LIN {X 0,Y 573.093,Z 391.869,A -85,B 0,C 180,E1 -2255.983,E2 -2255.983} C_VEL
LIN {X 0,Y 573.103,Z 385.471,A -85,B 0,C 180,E1 -2257.043,E2 -2257.043} C_VEL
LIN {X 0,Y 573.177,Z 377.482,A -85,B 0,C 180,E1 -2258.106,E2 -2258.106} C_VEL
LIN {X 0,Y 573.253,Z 369.34,A -85,B 0,C 180,E1 -2258.992,E2 -2258.992} C_VEL
LIN {X 0,Y 573.348,Z 359.406,A -85,B 0,C 180,E1 -2259.881,E2 -2259.881} C_VEL
LIN {X 0,Y 573.512,Z 348.221,A -85,B 0,C 180,E1 -2260.679,E2 -2260.679} C_VEL
LIN {X 0,Y 573.585,Z 337.185,A -85,B 0,C 180,E1 -2261.305,E2 -2261.305} C_VEL
LIN {X 0,Y 573.699,Z 324.995,A -85,B 0,C 180,E1 -2261.84,E2 -2261.84} C_VEL
LIN {X 0,Y 573.829,Z 312.198,A -85,B 0,C 180,E1 -2262.241,E2 -2262.241} C_VEL
LIN {X 0,Y 573.911,Z 300.143,A -85,B 0,C 180,E1 -2262.486,E2 -2262.486} C_VEL
LIN {X 0,Y 573.985,Z 198.766,A -85,B 0,C 180,E1 -2263.768,E2 -2263.768} C_VEL
LIN {X 0,Y 573.395,Z 194.617,A -85,B 0,C 180,E1 -2263.85,E2 -2263.85} C_VEL
LIN {X 0,Y 573.569,Z 174.135,A -85,B 0,C 180,E1 -2266.725,E2 -2266.725} C_VEL
LIN {X 0,Y 573.784,Z 153.422,A -85,B 0,C 180,E1 -2269.646,E2 -2269.646} C_VEL
LIN {X 0,Y 573.931,Z 133.412,A -85,B 0,C 180,E1 -2272.498,E2 -2272.498} C_VEL
LIN {X 0,Y 573.521,Z 128.586,A -85,B 0,C 180,E1 -2273.211,E2 -2273.211} C_VEL
LIN {X 0,Y 573.218,Z 127.086,A -85,B 0,C 180,E1 -2273.44,E2 -2273.44} C_VEL
LIN {X 0,Y 573.238,Z 127.079,A -85,B 0,C 180,E1 -2276.19,E2 -2276.19} C_VEL
LIN {X 0,Y 573.203,Z 127.08,A -85,B 0,C 180,E1 -2278.565,E2 -2278.565} C_VEL
LIN {X 0,Y 573.214,Z 127.08,A -85,B 0,C 180,E1 -2280.993,E2 -2280.993} C_VEL
LIN {X 0,Y 573.238,Z 127.084,A -85,B 0,C 180,E1 -2283.52,E2 -2283.52} C_VEL
LIN {X 0,Y 573.184,Z 127.083,A -85,B 0,C 180,E1 -2286.053,E2 -2286.053} C_VEL
LIN {X 0,Y 573.229,Z 127.077,A -85,B 0,C 180,E1 -2288.702,E2 -2288.702} C_VEL
LIN {X 0,Y 573.205,Z 127.084,A -85,B 0,C 180,E1 -2291.59,E2 -2291.59} C_VEL
LIN {X 0,Y 573.216,Z 127.077,A -85,B 0,C 180,E1 -2294.334,E2 -2294.334} C_VEL
LIN {X 0,Y 573.212,Z 127.084,A -85,B 0,C 180,E1 -2297.36,E2 -2297.36} C_VEL
LIN {X 0,Y 573.224,Z 127.077,A -85,B 0,C 180,E1 -2300.391,E2 -2300.391} C_VEL
LIN {X 0,Y 573.223,Z 127.085,A -85,B 0,C 180,E1 -2303.075,E2 -2303.075} C_VEL
LIN {X 0,Y 573.238,Z 127.075,A -85,B 0,C 180,E1 -2305.669,E2 -2305.669} C_VEL
LIN {X 0,Y 573.215,Z 127.078,A -85,B 0,C 180,E1 -2308.183,E2 -2308.183} C_VEL
LIN {X 0,Y 573.222,Z 127.084,A -85,B 0,C 180,E1 -2310.632,E2 -2310.632} C_VEL
LIN {X 0,Y 573.205,Z 127.079,A -85,B 0,C 180,E1 -2313.512,E2 -2313.512} C_VEL
LIN {X 0,Y 573.184,Z 127.084,A -85,B 0,C 180,E1 -2316.132,E2 -2316.132} C_VEL
LIN {X 0,Y 573.215,Z 127.079,A -85,B 0,C 180,E1 -2319.172,E2 -2319.172} C_VEL
LIN {X 0,Y 573.181,Z 127.082,A -85,B 0,C 180,E1 -2321.41,E2 -2321.41} C_VEL
LIN {X 0,Y 573.192,Z 127.089,A -85,B 0,C 180,E1 -2324.351,E2 -2324.351} C_VEL
LIN {X 0,Y 573.183,Z 127.088,A -85,B 0,C 180,E1 -2326.528,E2 -2326.528} C_VEL
LIN {X 0,Y 573.234,Z 127.075,A -85,B 0,C 180,E1 -2329.403,E2 -2329.403} C_VEL
LIN {X 0,Y 573.207,Z 127.087,A -85,B 0,C 180,E1 -2332.249,E2 -2332.249} C_VEL
LIN {X 0,Y 573.262,Z 127.071,A -85,B 0,C 180,E1 -2335.077,E2 -2335.077} C_VEL
LIN {X 0,Y 573.301,Z 127.074,A -85,B 0,C 180,E1 -2337.892,E2 -2337.892} C_VEL
LIN {X 0,Y 573.307,Z 127.075,A -85,B 0,C 180,E1 -2340,E2 -2340} C_VEL
LIN {X 0,Y 573.26,Z 127.072,A -85,B 0,C 180,E1 -2342.811,E2 -2342.811} C_VEL
LIN {X 0,Y 573.267,Z 127.078,A -85,B 0,C 180,E1 -2345.628,E2 -2345.628} C_VEL
LIN {X 0,Y 573.232,Z 127.076,A -85,B 0,C 180,E1 -2348.46,E2 -2348.46} C_VEL
LIN {X 0,Y 573.261,Z 127.076,A -85,B 0,C 180,E1 -2351.312,E2 -2351.312} C_VEL
LIN {X 0,Y 573.246,Z 127.074,A -85,B 0,C 180,E1 -2354.415,E2 -2354.415} C_VEL
LIN {X 0,Y 573.168,Z 127.087,A -85,B 0,C 180,E1 -2357.114,E2 -2357.114} C_VEL
LIN {X 0,Y 573.255,Z 127.081,A -85,B 0,C 180,E1 -2359.331,E2 -2359.331} C_VEL
LIN {X 0,Y 573.21,Z 127.078,A -85,B 0,C 180,E1 -2362.339,E2 -2362.339} C_VEL
LIN {X 0,Y 573.187,Z 127.081,A -85,B 0,C 180,E1 -2364.347,E2 -2364.347} C_VEL
LIN {X 0,Y 572.548,Z 127.166,A -85,B 0,C 180,E1 -2364.933,E2 -2364.933} C_VEL
LIN {X 0,Y 569.719,Z 127.523,A -85,B 0,C 180,E1 -2365.885,E2 -2365.885} C_VEL
LIN {X 0,Y 567.301,Z 127.827,A -85,B 0,C 180,E1 -2366.65,E2 -2366.65} C_VEL
LIN {X 0,Y 566.245,Z 127.955,A -85,B 0,C 180,E1 -2367.242,E2 -2367.242} C_VEL
LIN {X 0,Y 566.15,Z 127.963,A -85,B 0,C 180,E1 -2367.442,E2 -2367.442} C_VEL
LIN {X 0,Y 566.159,Z 127.958,A -85,B 0,C 180,E1 -2369.771,E2 -2369.771} C_VEL
LIN {X 0,Y 566.184,Z 127.954,A -85,B 0,C 180,E1 -2372.429,E2 -2372.429} C_VEL
LIN {X 0,Y 566.168,Z 127.965,A -85,B 0,C 180,E1 -2374.99,E2 -2374.99} C_VEL
LIN {X 0,Y 566.187,Z 127.955,A -85,B 0,C 180,E1 -2377.462,E2 -2377.462} C_VEL
LIN {X 0,Y 566.199,Z 127.953,A -85,B 0,C 180,E1 -2380.2,E2 -2380.2} C_VEL
LIN {X 0,Y 566.174,Z 127.959,A -85,B 0,C 180,E1 -2383.057,E2 -2383.057} C_VEL
LIN {X 0,Y 566.187,Z 127.954,A -85,B 0,C 180,E1 -2386.05,E2 -2386.05} C_VEL
LIN {X 0,Y 566.199,Z 127.953,A -85,B 0,C 180,E1 -2389.216,E2 -2389.216} C_VEL
LIN {X 0,Y 566.175,Z 127.954,A -85,B 0,C 180,E1 -2391.637,E2 -2391.637} C_VEL
LIN {X 0,Y 566.145,Z 127.965,A -85,B 0,C 180,E1 -2394.308,E2 -2394.308} C_VEL
LIN {X 0,Y 566.206,Z 127.953,A -85,B 0,C 180,E1 -2396.898,E2 -2396.898} C_VEL
LIN {X 0,Y 566.167,Z 127.955,A -85,B 0,C 180,E1 -2399.407,E2 -2399.407} C_VEL
LIN {X 0,Y 566.186,Z 127.957,A -85,B 0,C 180,E1 -2401.857,E2 -2401.857} C_VEL
LIN {X 0,Y 566.194,Z 127.961,A -85,B 0,C 180,E1 -2404.251,E2 -2404.251} C_VEL
LIN {X 0,Y 566.17,Z 127.956,A -85,B 0,C 180,E1 -2407.369,E2 -2407.369} C_VEL
LIN {X 0,Y 566.202,Z 127.957,A -85,B 0,C 180,E1 -2409.663,E2 -2409.663} C_VEL
LIN {X 0,Y 566.225,Z 128.065,A -85,B 0,C 180,E1 -2410.877,E2 -2410.877} C_VEL
LIN {X 0,Y 566.465,Z 134.818,A -85,B 0,C 180,E1 -2412.118,E2 -2412.118} C_VEL
LIN {X 0,Y 566.294,Z 150.062,A -85,B 0,C 180,E1 -2414.894,E2 -2414.894} C_VEL
LIN {X 0,Y 566.255,Z 156.422,A -85,B 0,C 180,E1 -2416.055,E2 -2416.055} C_VEL
LIN {X 0,Y 567.161,Z 162.399,A -85,B 0,C 180,E1 -2416.155,E2 -2416.155} C_VEL
LIN {X 0,Y 566.967,Z 262.997,A -85,B 0,C 180,E1 -2417.449,E2 -2417.449} C_VEL
LIN {X 0,Y 566.83,Z 276.241,A -85,B 0,C 180,E1 -2417.764,E2 -2417.764} C_VEL
LIN {X 0,Y 566.736,Z 288.394,A -85,B 0,C 180,E1 -2418.194,E2 -2418.194} C_VEL
LIN {X 0,Y 566.611,Z 300.586,A -85,B 0,C 180,E1 -2418.777,E2 -2418.777} C_VEL
LIN {X 0,Y 566.448,Z 311.561,A -85,B 0,C 180,E1 -2419.456,E2 -2419.456} C_VEL
LIN {X 0,Y 566.326,Z 322.078,A -85,B 0,C 180,E1 -2420.266,E2 -2420.266} C_VEL
LIN {X 0,Y 566.221,Z 330.674,A -85,B 0,C 180,E1 -2421.075,E2 -2421.075} C_VEL
LIN {X 0,Y 566.112,Z 338.594,A -85,B 0,C 180,E1 -2421.972,E2 -2421.972} C_VEL
LIN {X 0,Y 566.049,Z 345.161,A -85,B 0,C 180,E1 -2422.868,E2 -2422.868} C_VEL
LIN {X 0,Y 566.003,Z 351.63,A -85,B 0,C 180,E1 -2423.942,E2 -2423.942} C_VEL
LIN {X 0,Y 565.877,Z 356.766,A -85,B 0,C 180,E1 -2425.013,E2 -2425.013} C_VEL
LIN {X 0,Y 565.926,Z 360.755,A -85,B 0,C 180,E1 -2426.084,E2 -2426.084} C_VEL
LIN {X 0,Y 565.877,Z 363.704,A -85,B 0,C 180,E1 -2427.153,E2 -2427.153} C_VEL
LIN {X 0,Y 565.841,Z 365.127,A -85,B 0,C 180,E1 -2427.865,E2 -2427.865} C_VEL
LIN {X 0,Y 565.841,Z 366.757,A -85,B 0,C 180,E1 -2429.289,E2 -2429.289} C_VEL
LIN {X 0,Y 565.839,Z 366.996,A -85,B 0,C 180,E1 -2430,E2 -2430} C_VEL
LIN {X 0,Y 565.841,Z 366.815,A -85,B 0,C 180,E1 -2430.712,E2 -2430.712} C_VEL
LIN {X 0,Y 565.841,Z 365.266,A -85,B 0,C 180,E1 -2432.136,E2 -2432.136} C_VEL
LIN {X 0,Y 565.878,Z 363.905,A -85,B 0,C 180,E1 -2432.848,E2 -2432.848} C_VEL
LIN {X 0,Y 565.927,Z 361.028,A -85,B 0,C 180,E1 -2433.917,E2 -2433.917} C_VEL
LIN {X 0,Y 565.878,Z 357.128,A -85,B 0,C 180,E1 -2434.988,E2 -2434.988} C_VEL
LIN {X 0,Y 565.991,Z 352.096,A -85,B 0,C 180,E1 -2436.059,E2 -2436.059} C_VEL
LIN {X 0,Y 566.031,Z 345.77,A -85,B 0,C 180,E1 -2437.133,E2 -2437.133} C_VEL
LIN {X 0,Y 566.128,Z 337.847,A -85,B 0,C 180,E1 -2438.208,E2 -2438.208} C_VEL
LIN {X 0,Y 566.249,Z 327.995,A -85,B 0,C 180,E1 -2439.285,E2 -2439.285} C_VEL
LIN {X 0,Y 566.424,Z 317.675,A -85,B 0,C 180,E1 -2440.184,E2 -2440.184} C_VEL
LIN {X 0,Y 566.507,Z 306.391,A -85,B 0,C 180,E1 -2440.973,E2 -2440.973} C_VEL
LIN {X 0,Y 566.691,Z 295.182,A -85,B 0,C 180,E1 -2441.592,E2 -2441.592} C_VEL
LIN {X 0,Y 566.788,Z 282.587,A -85,B 0,C 180,E1 -2442.119,E2 -2442.119} C_VEL
LIN {X 0,Y 566.93,Z 269.409,A -85,B 0,C 180,E1 -2442.507,E2 -2442.507} C_VEL
LIN {X 0,Y 567.04,Z 257.034,A -85,B 0,C 180,E1 -2442.732,E2 -2442.732} C_VEL
LIN {X 0,Y 567.066,Z 161.334,A -85,B 0,C 180,E1 -2443.951,E2 -2443.951} C_VEL
LIN {X 0,Y 566.237,Z 156.331,A -85,B 0,C 180,E1 -2444.052,E2 -2444.052} C_VEL
LIN {X 0,Y 566.391,Z 140.839,A -85,B 0,C 180,E1 -2446.877,E2 -2446.877} C_VEL
LIN {X 0,Y 566.442,Z 130.18,A -85,B 0,C 180,E1 -2448.82,E2 -2448.82} C_VEL
LIN {X 0,Y 566.223,Z 127.955,A -85,B 0,C 180,E1 -2449.251,E2 -2449.251} C_VEL
LIN {X 0,Y 566.189,Z 127.961,A -85,B 0,C 180,E1 -2451.863,E2 -2451.863} C_VEL
LIN {X 0,Y 566.185,Z 127.954,A -85,B 0,C 180,E1 -2455.022,E2 -2455.022} C_VEL
LIN {X 0,Y 566.173,Z 127.957,A -85,B 0,C 180,E1 -2457.341,E2 -2457.341} C_VEL
LIN {X 0,Y 566.173,Z 127.964,A -85,B 0,C 180,E1 -2459.77,E2 -2459.77} C_VEL
LIN {X 0,Y 566.201,Z 127.952,A -85,B 0,C 180,E1 -2462.429,E2 -2462.429} C_VEL
LIN {X 0,Y 566.178,Z 127.955,A -85,B 0,C 180,E1 -2464.989,E2 -2464.989} C_VEL
LIN {X 0,Y 566.192,Z 127.96,A -85,B 0,C 180,E1 -2467.461,E2 -2467.461} C_VEL
LIN {X 0,Y 566.206,Z 127.951,A -85,B 0,C 180,E1 -2470.199,E2 -2470.199} C_VEL
LIN {X 0,Y 566.192,Z 127.956,A -85,B 0,C 180,E1 -2473.055,E2 -2473.055} C_VEL
LIN {X 0,Y 566.157,Z 127.957,A -85,B 0,C 180,E1 -2476.053,E2 -2476.053} C_VEL
LIN {X 0,Y 566.165,Z 127.959,A -85,B 0,C 180,E1 -2478.859,E2 -2478.859} C_VEL
LIN {X 0,Y 566.202,Z 127.956,A -85,B 0,C 180,E1 -2481.443,E2 -2481.443} C_VEL
LIN {X 0,Y 566.141,Z 127.959,A -85,B 0,C 180,E1 -2484.306,E2 -2484.306} C_VEL
LIN {X 0,Y 566.192,Z 127.96,A -85,B 0,C 180,E1 -2486.896,E2 -2486.896} C_VEL
LIN {X 0,Y 566.159,Z 127.959,A -85,B 0,C 180,E1 -2489.406,E2 -2489.406} C_VEL
LIN {X 0,Y 566.147,Z 127.958,A -85,B 0,C 180,E1 -2491.854,E2 -2491.854} C_VEL
LIN {X 0,Y 566.197,Z 127.954,A -85,B 0,C 180,E1 -2494.25,E2 -2494.25} C_VEL
LIN {X 0,Y 566.158,Z 127.958,A -85,B 0,C 180,E1 -2497.367,E2 -2497.367} C_VEL
LIN {X 0,Y 566.194,Z 127.952,A -85,B 0,C 180,E1 -2499.662,E2 -2499.662} C_VEL
LIN {X 0,Y 566.161,Z 127.957,A -85,B 0,C 180,E1 -2501.92,E2 -2501.92} C_VEL
LIN {X 0,Y 566.176,Z 127.958,A -85,B 0,C 180,E1 -2504.89,E2 -2504.89} C_VEL
LIN {X 0,Y 566.173,Z 127.956,A -85,B 0,C 180,E1 -2507.818,E2 -2507.818} C_VEL
LIN {X 0,Y 566.163,Z 127.96,A -85,B 0,C 180,E1 -2509.992,E2 -2509.992} C_VEL
LIN {X 0,Y 566.178,Z 127.956,A -85,B 0,C 180,E1 -2512.869,E2 -2512.869} C_VEL
LIN {X 0,Y 566.246,Z 127.946,A -85,B 0,C 180,E1 -2515.016,E2 -2515.016} C_VEL
LIN {X 0,Y 566.274,Z 127.947,A -85,B 0,C 180,E1 -2517.866,E2 -2517.866} C_VEL
LIN {X 0,Y 566.281,Z 127.95,A -85,B 0,C 180,E1 -2520,E2 -2520} C_VEL
LIN {X 0,Y 566.232,Z 127.947,A -85,B 0,C 180,E1 -2522.846,E2 -2522.846} C_VEL
LIN {X 0,Y 566.229,Z 127.954,A -85,B 0,C 180,E1 -2525.699,E2 -2525.699} C_VEL
LIN {X 0,Y 566.178,Z 127.955,A -85,B 0,C 180,E1 -2528.566,E2 -2528.566} C_VEL
LIN {X 0,Y 566.187,Z 127.958,A -85,B 0,C 180,E1 -2531.455,E2 -2531.455} C_VEL
LIN {X 0,Y 566.178,Z 127.954,A -85,B 0,C 180,E1 -2534.486,E2 -2534.486} C_VEL
LIN {X 0,Y 566.152,Z 127.963,A -85,B 0,C 180,E1 -2537.333,E2 -2537.333} C_VEL
LIN {X 0,Y 566.169,Z 127.964,A -85,B 0,C 180,E1 -2539.582,E2 -2539.582} C_VEL
LIN {X 0,Y 566.141,Z 127.962,A -85,B 0,C 180,E1 -2541.865,E2 -2541.865} C_VEL
LIN {X 0,Y 566.147,Z 127.958,A -85,B 0,C 180,E1 -2544.183,E2 -2544.183} C_VEL
LIN {X 0,Y 566.17,Z 127.956,A -85,B 0,C 180,E1 -2546.652,E2 -2546.652} C_VEL
LIN {X 0,Y 566.143,Z 127.96,A -85,B 0,C 180,E1 -2549.772,E2 -2549.772} C_VEL
LIN {X 0,Y 566.188,Z 127.953,A -85,B 0,C 180,E1 -2552.428,E2 -2552.428} C_VEL
LIN {X 0,Y 566.16,Z 127.964,A -85,B 0,C 180,E1 -2554.987,E2 -2554.987} C_VEL
LIN {X 0,Y 566.188,Z 127.956,A -85,B 0,C 180,E1 -2557.462,E2 -2557.462} C_VEL
LIN {X 0,Y 566.203,Z 127.952,A -85,B 0,C 180,E1 -2560.2,E2 -2560.2} C_VEL
LIN {X 0,Y 566.177,Z 127.96,A -85,B 0,C 180,E1 -2563.057,E2 -2563.057} C_VEL
LIN {X 0,Y 566.155,Z 127.958,A -85,B 0,C 180,E1 -2566.054,E2 -2566.054} C_VEL
LIN {X 0,Y 566.163,Z 127.963,A -85,B 0,C 180,E1 -2568.86,E2 -2568.86} C_VEL
LIN {X 0,Y 566.198,Z 127.952,A -85,B 0,C 180,E1 -2571.444,E2 -2571.444} C_VEL
LIN {X 0,Y 566.141,Z 127.965,A -85,B 0,C 180,E1 -2574.306,E2 -2574.306} C_VEL
LIN {X 0,Y 566.195,Z 127.955,A -85,B 0,C 180,E1 -2576.896,E2 -2576.896} C_VEL
LIN {X 0,Y 566.168,Z 127.956,A -85,B 0,C 180,E1 -2579.407,E2 -2579.407} C_VEL
LIN {X 0,Y 566.171,Z 127.959,A -85,B 0,C 180,E1 -2581.855,E2 -2581.855} C_VEL
LIN {X 0,Y 566.194,Z 127.962,A -85,B 0,C 180,E1 -2584.25,E2 -2584.25} C_VEL
LIN {X 0,Y 566.179,Z 128.025,A -85,B 0,C 180,E1 -2586.426,E2 -2586.426} C_VEL
LIN {X 0,Y 567.021,Z 133.161,A -85,B 0,C 180,E1 -2587.211,E2 -2587.211} C_VEL
LIN {X 0,Y 566.812,Z 152.9,A -85,B 0,C 180,E1 -2590.064,E2 -2590.064} C_VEL
LIN {X 0,Y 566.588,Z 174.338,A -85,B 0,C 180,E1 -2593.111,E2 -2593.111} C_VEL
LIN {X 0,Y 566.39,Z 194.612,A -85,B 0,C 180,E1 -2595.974,E2 -2595.974} C_VEL
LIN {X 0,Y 567.155,Z 200.495,A -85,B 0,C 180,E1 -2596.085,E2 -2596.085} C_VEL
LIN {X 0,Y 566.961,Z 302.936,A -85,B 0,C 180,E1 -2597.403,E2 -2597.403} C_VEL
LIN {X 0,Y 566.84,Z 316.211,A -85,B 0,C 180,E1 -2597.718,E2 -2597.718} C_VEL
LIN {X 0,Y 566.743,Z 328.373,A -85,B 0,C 180,E1 -2598.148,E2 -2598.148} C_VEL
LIN {X 0,Y 566.604,Z 340.235,A -85,B 0,C 180,E1 -2598.712,E2 -2598.712} C_VEL
LIN {X 0,Y 566.439,Z 352.192,A -85,B 0,C 180,E1 -2599.455,E2 -2599.455} C_VEL
LIN {X 0,Y 566.325,Z 362.602,A -85,B 0,C 180,E1 -2600.265,E2 -2600.265} C_VEL
LIN {X 0,Y 566.207,Z 371.111,A -85,B 0,C 180,E1 -2601.074,E2 -2601.074} C_VEL
LIN {X 0,Y 566.112,Z 378.958,A -85,B 0,C 180,E1 -2601.971,E2 -2601.971} C_VEL
LIN {X 0,Y 566.004,Z 386.621,A -85,B 0,C 180,E1 -2603.046,E2 -2603.046} C_VEL
LIN {X 0,Y 566.004,Z 393.678,A -85,B 0,C 180,E1 -2604.299,E2 -2604.299} C_VEL
LIN {X 0,Y 565.933,Z 398.371,A -85,B 0,C 180,E1 -2605.37,E2 -2605.37} C_VEL
LIN {X 0,Y 565.927,Z 401.957,A -85,B 0,C 180,E1 -2606.44,E2 -2606.44} C_VEL
LIN {X 0,Y 565.878,Z 403.807,A -85,B 0,C 180,E1 -2607.152,E2 -2607.152} C_VEL
LIN {X 0,Y 565.846,Z 406.183,A -85,B 0,C 180,E1 -2608.576,E2 -2608.576} C_VEL
LIN {X 0,Y 565.839,Z 407,A -85,B 0,C 180,E1 -2610,E2 -2610} C_VEL
LIN {X 0,Y 565.846,Z 406.185,A -85,B 0,C 180,E1 -2611.423,E2 -2611.423} C_VEL
LIN {X 0,Y 565.878,Z 403.811,A -85,B 0,C 180,E1 -2612.847,E2 -2612.847} C_VEL
LIN {X 0,Y 565.926,Z 400.897,A -85,B 0,C 180,E1 -2613.916,E2 -2613.916} C_VEL
LIN {X 0,Y 565.878,Z 396.95,A -85,B 0,C 180,E1 -2614.987,E2 -2614.987} C_VEL
LIN {X 0,Y 566.004,Z 391.87,A -85,B 0,C 180,E1 -2616.058,E2 -2616.058} C_VEL
LIN {X 0,Y 566.04,Z 385.471,A -85,B 0,C 180,E1 -2617.132,E2 -2617.132} C_VEL
LIN {X 0,Y 566.133,Z 377.482,A -85,B 0,C 180,E1 -2618.207,E2 -2618.207} C_VEL
LIN {X 0,Y 566.228,Z 369.339,A -85,B 0,C 180,E1 -2619.105,E2 -2619.105} C_VEL
LIN {X 0,Y 566.347,Z 359.405,A -85,B 0,C 180,E1 -2620.004,E2 -2620.004} C_VEL
LIN {X 0,Y 566.535,Z 348.299,A -85,B 0,C 180,E1 -2620.807,E2 -2620.807} C_VEL
LIN {X 0,Y 566.611,Z 337.183,A -85,B 0,C 180,E1 -2621.446,E2 -2621.446} C_VEL
LIN {X 0,Y 566.744,Z 324.992,A -85,B 0,C 180,E1 -2621.987,E2 -2621.987} C_VEL
LIN {X 0,Y 566.913,Z 312.197,A -85,B 0,C 180,E1 -2622.393,E2 -2622.393} C_VEL
LIN {X 0,Y 567.006,Z 300.142,A -85,B 0,C 180,E1 -2622.641,E2 -2622.641} C_VEL
LIN {X 0,Y 567.051,Z 199.325,A -85,B 0,C 180,E1 -2623.932,E2 -2623.932} C_VEL
LIN {X 0,Y 566.39,Z 194.617,A -85,B 0,C 180,E1 -2624.025,E2 -2624.025} C_VEL
LIN {X 0,Y 566.588,Z 174.314,A -85,B 0,C 180,E1 -2626.892,E2 -2626.892} C_VEL
LIN {X 0,Y 566.853,Z 151.591,A -85,B 0,C 180,E1 -2630.123,E2 -2630.123} C_VEL
LIN {X 0,Y 566.992,Z 133.166,A -85,B 0,C 180,E1 -2632.789,E2 -2632.789} C_VEL
LIN {X 0,Y 566.196,Z 127.961,A -85,B 0,C 180,E1 -2633.597,E2 -2633.597} C_VEL
LIN {X 0,Y 566.187,Z 127.955,A -85,B 0,C 180,E1 -2636.542,E2 -2636.542} C_VEL
LIN {X 0,Y 566.161,Z 127.958,A -85,B 0,C 180,E1 -2638.954,E2 -2638.954} C_VEL
LIN {X 0,Y 566.18,Z 127.961,A -85,B 0,C 180,E1 -2641.422,E2 -2641.422} C_VEL
LIN {X 0,Y 566.191,Z 127.956,A -85,B 0,C 180,E1 -2643.956,E2 -2643.956} C_VEL
LIN {X 0,Y 566.176,Z 127.954,A -85,B 0,C 180,E1 -2646.571,E2 -2646.571} C_VEL
LIN {X 0,Y 566.204,Z 127.955,A -85,B 0,C 180,E1 -2649.684,E2 -2649.684} C_VEL
LIN {X 0,Y 566.165,Z 127.956,A -85,B 0,C 180,E1 -2652.09,E2 -2652.09} C_VEL
LIN {X 0,Y 566.158,Z 127.962,A -85,B 0,C 180,E1 -2654.962,E2 -2654.962} C_VEL
LIN {X 0,Y 566.163,Z 127.956,A -85,B 0,C 180,E1 -2657.908,E2 -2657.908} C_VEL
LIN {X 0,Y 566.2,Z 127.956,A -85,B 0,C 180,E1 -2660.725,E2 -2660.725} C_VEL
LIN {X 0,Y 566.172,Z 127.958,A -85,B 0,C 180,E1 -2663.428,E2 -2663.428} C_VEL
LIN {X 0,Y 566.187,Z 127.954,A -85,B 0,C 180,E1 -2666.268,E2 -2666.268} C_VEL
LIN {X 0,Y 566.172,Z 127.963,A -85,B 0,C 180,E1 -2668.925,E2 -2668.925} C_VEL
LIN {X 0,Y 566.139,Z 127.959,A -85,B 0,C 180,E1 -2671.853,E2 -2671.853} C_VEL
LIN {X 0,Y 566.181,Z 127.957,A -85,B 0,C 180,E1 -2674.249,E2 -2674.249} C_VEL
LIN {X 0,Y 566.135,Z 127.96,A -85,B 0,C 180,E1 -2677.367,E2 -2677.367} C_VEL
LIN {X 0,Y 566.158,Z 127.957,A -85,B 0,C 180,E1 -2679.661,E2 -2679.661} C_VEL
LIN {X 0,Y 566.151,Z 127.959,A -85,B 0,C 180,E1 -2681.92,E2 -2681.92} C_VEL
LIN {X 0,Y 566.168,Z 127.958,A -85,B 0,C 180,E1 -2684.89,E2 -2684.89} C_VEL
LIN {X 0,Y 566.166,Z 127.958,A -85,B 0,C 180,E1 -2687.817,E2 -2687.817} C_VEL
LIN {X 0,Y 566.151,Z 127.963,A -85,B 0,C 180,E1 -2689.992,E2 -2689.992} C_VEL
LIN {X 0,Y 566.17,Z 127.956,A -85,B 0,C 180,E1 -2692.869,E2 -2692.869} C_VEL
LIN {X 0,Y 566.238,Z 127.947,A -85,B 0,C 180,E1 -2695.016,E2 -2695.016} C_VEL
LIN {X 0,Y 566.27,Z 127.95,A -85,B 0,C 180,E1 -2697.866,E2 -2697.866} C_VEL
LIN {X 0,Y 566.275,Z 127.951,A -85,B 0,C 180,E1 -2700,E2 -2700} C_VEL
LIN {X 0,Y 566.228,Z 127.948,A -85,B 0,C 180,E1 -2702.846,E2 -2702.846} C_VEL
LIN {X 0,Y 566.236,Z 127.955,A -85,B 0,C 180,E1 -2705.699,E2 -2705.699} C_VEL
LIN {X 0,Y 566.183,Z 127.953,A -85,B 0,C 180,E1 -2708.566,E2 -2708.566} C_VEL
LIN {X 0,Y 566.228,Z 127.954,A -85,B 0,C 180,E1 -2711.455,E2 -2711.455} C_VEL
LIN {X 0,Y 566.202,Z 127.951,A -85,B 0,C 180,E1 -2714.498,E2 -2714.498} C_VEL
LIN {X 0,Y 566.141,Z 127.966,A -85,B 0,C 180,E1 -2717.334,E2 -2717.334} C_VEL
LIN {X 0,Y 566.188,Z 127.96,A -85,B 0,C 180,E1 -2719.582,E2 -2719.582} C_VEL
LIN {X 0,Y 566.176,Z 127.957,A -85,B 0,C 180,E1 -2721.863,E2 -2721.863} C_VEL
LIN {X 0,Y 566.168,Z 127.961,A -85,B 0,C 180,E1 -2725.022,E2 -2725.022} C_VEL
LIN {X 0,Y 566.15,Z 127.963,A -85,B 0,C 180,E1 -2727.442,E2 -2727.442} C_VEL
LIN {X 0,Y 565.461,Z 128.046,A -85,B 0,C 180,E1 -2728.036,E2 -2728.036} C_VEL
LIN {X 0,Y 562.605,Z 128.406,A -85,B 0,C 180,E1 -2729,E2 -2729} C_VEL
LIN {X 0,Y 560.213,Z 128.7,A -85,B 0,C 180,E1 -2729.776,E2 -2729.776} C_VEL
LIN {X 0,Y 559.196,Z 128.825,A -85,B 0,C 180,E1 -2730.374,E2 -2730.374} C_VEL
LIN {X 0,Y 559.118,Z 128.836,A -85,B 0,C 180,E1 -2730.577,E2 -2730.577} C_VEL
LIN {X 0,Y 559.139,Z 128.835,A -85,B 0,C 180,E1 -2732.717,E2 -2732.717} C_VEL
LIN {X 0,Y 559.118,Z 128.838,A -85,B 0,C 180,E1 -2735.325,E2 -2735.325} C_VEL
LIN {X 0,Y 559.121,Z 128.833,A -85,B 0,C 180,E1 -2738.019,E2 -2738.019} C_VEL
LIN {X 0,Y 559.146,Z 128.84,A -85,B 0,C 180,E1 -2740.814,E2 -2740.814} C_VEL
LIN {X 0,Y 559.102,Z 128.835,A -85,B 0,C 180,E1 -2743.738,E2 -2743.738} C_VEL
LIN {X 0,Y 559.13,Z 128.835,A -85,B 0,C 180,E1 -2746.266,E2 -2746.266} C_VEL
LIN {X 0,Y 559.15,Z 128.831,A -85,B 0,C 180,E1 -2749.188,E2 -2749.188} C_VEL
LIN {X 0,Y 559.123,Z 128.835,A -85,B 0,C 180,E1 -2751.983,E2 -2751.983} C_VEL
LIN {X 0,Y 559.124,Z 128.837,A -85,B 0,C 180,E1 -2754.789,E2 -2754.789} C_VEL
LIN {X 0,Y 559.151,Z 128.829,A -85,B 0,C 180,E1 -2757.366,E2 -2757.366} C_VEL
LIN {X 0,Y 559.119,Z 128.841,A -85,B 0,C 180,E1 -2760.149,E2 -2760.149} C_VEL
LIN {X 0,Y 559.14,Z 128.831,A -85,B 0,C 180,E1 -2763.179,E2 -2763.179} C_VEL
LIN {X 0,Y 559.123,Z 128.834,A -85,B 0,C 180,E1 -2765.494,E2 -2765.494} C_VEL
LIN {X 0,Y 559.171,Z 128.831,A -85,B 0,C 180,E1 -2768.625,E2 -2768.625} C_VEL
LIN {X 0,Y 559.209,Z 128.962,A -85,B 0,C 180,E1 -2770.793,E2 -2770.793} C_VEL
LIN {X 0,Y 559.453,Z 135.875,A -85,B 0,C 180,E1 -2772.075,E2 -2772.075} C_VEL
LIN {X 0,Y 559.295,Z 152.435,A -85,B 0,C 180,E1 -2775.11,E2 -2775.11} C_VEL
LIN {X 0,Y 559.243,Z 156.672,A -85,B 0,C 180,E1 -2775.876,E2 -2775.876} C_VEL
LIN {X 0,Y 560.255,Z 162.655,A -85,B 0,C 180,E1 -2775.981,E2 -2775.981} C_VEL
LIN {X 0,Y 560.051,Z 263.136,A -85,B 0,C 180,E1 -2777.292,E2 -2777.292} C_VEL
LIN {X 0,Y 559.899,Z 276.352,A -85,B 0,C 180,E1 -2777.611,E2 -2777.611} C_VEL
LIN {X 0,Y 559.784,Z 288.472,A -85,B 0,C 180,E1 -2778.045,E2 -2778.045} C_VEL
LIN {X 0,Y 559.648,Z 300.124,A -85,B 0,C 180,E1 -2778.607,E2 -2778.607} C_VEL
LIN {X 0,Y 559.473,Z 311.566,A -85,B 0,C 180,E1 -2779.323,E2 -2779.323} C_VEL
LIN {X 0,Y 559.307,Z 322.083,A -85,B 0,C 180,E1 -2780.143,E2 -2780.143} C_VEL
LIN {X 0,Y 559.196,Z 330.679,A -85,B 0,C 180,E1 -2780.962,E2 -2780.962} C_VEL
LIN {X 0,Y 559.05,Z 338.599,A -85,B 0,C 180,E1 -2781.87,E2 -2781.87} C_VEL
LIN {X 0,Y 558.971,Z 346.46,A -85,B 0,C 180,E1 -2782.977,E2 -2782.977} C_VEL
LIN {X 0,Y 558.936,Z 353.456,A -85,B 0,C 180,E1 -2784.227,E2 -2784.227} C_VEL
LIN {X 0,Y 558.826,Z 358.196,A -85,B 0,C 180,E1 -2785.312,E2 -2785.312} C_VEL
LIN {X 0,Y 558.836,Z 361.829,A -85,B 0,C 180,E1 -2786.395,E2 -2786.395} C_VEL
LIN {X 0,Y 558.799,Z 363.706,A -85,B 0,C 180,E1 -2787.117,E2 -2787.117} C_VEL
LIN {X 0,Y 558.747,Z 365.127,A -85,B 0,C 180,E1 -2787.838,E2 -2787.838} C_VEL
LIN {X 0,Y 558.741,Z 366.757,A -85,B 0,C 180,E1 -2789.28,E2 -2789.28} C_VEL
LIN {X 0,Y 558.74,Z 366.996,A -85,B 0,C 180,E1 -2790,E2 -2790} C_VEL
LIN {X 0,Y 558.741,Z 366.815,A -85,B 0,C 180,E1 -2790.721,E2 -2790.721} C_VEL
LIN {X 0,Y 558.747,Z 365.263,A -85,B 0,C 180,E1 -2792.163,E2 -2792.163} C_VEL
LIN {X 0,Y 558.8,Z 363.903,A -85,B 0,C 180,E1 -2792.884,E2 -2792.884} C_VEL
LIN {X 0,Y 558.844,Z 361.026,A -85,B 0,C 180,E1 -2793.967,E2 -2793.967} C_VEL
LIN {X 0,Y 558.798,Z 357.125,A -85,B 0,C 180,E1 -2795.051,E2 -2795.051} C_VEL
LIN {X 0,Y 558.91,Z 352.093,A -85,B 0,C 180,E1 -2796.136,E2 -2796.136} C_VEL
LIN {X 0,Y 558.973,Z 345.766,A -85,B 0,C 180,E1 -2797.223,E2 -2797.223} C_VEL
LIN {X 0,Y 559.091,Z 337.842,A -85,B 0,C 180,E1 -2798.312,E2 -2798.312} C_VEL
LIN {X 0,Y 559.224,Z 327.988,A -85,B 0,C 180,E1 -2799.403,E2 -2799.403} C_VEL
LIN {X 0,Y 559.429,Z 317.666,A -85,B 0,C 180,E1 -2800.313,E2 -2800.313} C_VEL
LIN {X 0,Y 559.53,Z 306.643,A -85,B 0,C 180,E1 -2801.095,E2 -2801.095} C_VEL
LIN {X 0,Y 559.712,Z 296.488,A -85,B 0,C 180,E1 -2801.672,E2 -2801.672} C_VEL
LIN {X 0,Y 559.815,Z 285.029,A -85,B 0,C 180,E1 -2802.185,E2 -2802.185} C_VEL
LIN {X 0,Y 559.982,Z 272.23,A -85,B 0,C 180,E1 -2802.595,E2 -2802.595} C_VEL
LIN {X 0,Y 560.104,Z 260.133,A -85,B 0,C 180,E1 -2802.846,E2 -2802.846} C_VEL
LIN {X 0,Y 560.149,Z 161.747,A -85,B 0,C 180,E1 -2804.124,E2 -2804.124} C_VEL
LIN {X 0,Y 559.227,Z 156.524,A -85,B 0,C 180,E1 -2804.232,E2 -2804.232} C_VEL
LIN {X 0,Y 559.379,Z 141.188,A -85,B 0,C 180,E1 -2807.04,E2 -2807.04} C_VEL
LIN {X 0,Y 559.357,Z 130.178,A -85,B 0,C 180,E1 -2809.067,E2 -2809.067} C_VEL
LIN {X 0,Y 559.186,Z 128.832,A -85,B 0,C 180,E1 -2809.35,E2 -2809.35} C_VEL
LIN {X 0,Y 559.137,Z 128.839,A -85,B 0,C 180,E1 -2812.153,E2 -2812.153} C_VEL
LIN {X 0,Y 559.144,Z 128.831,A -85,B 0,C 180,E1 -2815.178,E2 -2815.178} C_VEL
LIN {X 0,Y 559.129,Z 128.839,A -85,B 0,C 180,E1 -2817.715,E2 -2817.715} C_VEL
LIN {X 0,Y 559.139,Z 128.834,A -85,B 0,C 180,E1 -2820.184,E2 -2820.184} C_VEL
LIN {X 0,Y 559.155,Z 128.829,A -85,B 0,C 180,E1 -2822.715,E2 -2822.715} C_VEL
LIN {X 0,Y 559.123,Z 128.837,A -85,B 0,C 180,E1 -2825.324,E2 -2825.324} C_VEL
LIN {X 0,Y 559.128,Z 128.835,A -85,B 0,C 180,E1 -2828.018,E2 -2828.018} C_VEL
LIN {X 0,Y 559.155,Z 128.83,A -85,B 0,C 180,E1 -2830.812,E2 -2830.812} C_VEL
LIN {X 0,Y 559.135,Z 128.836,A -85,B 0,C 180,E1 -2833.734,E2 -2833.734} C_VEL
LIN {X 0,Y 559.13,Z 128.834,A -85,B 0,C 180,E1 -2836.805,E2 -2836.805} C_VEL
LIN {X 0,Y 559.152,Z 128.838,A -85,B 0,C 180,E1 -2839.187,E2 -2839.187} C_VEL
LIN {X 0,Y 559.125,Z 128.833,A -85,B 0,C 180,E1 -2841.982,E2 -2841.982} C_VEL
LIN {X 0,Y 559.121,Z 128.838,A -85,B 0,C 180,E1 -2844.788,E2 -2844.788} C_VEL
LIN {X 0,Y 559.146,Z 128.834,A -85,B 0,C 180,E1 -2847.366,E2 -2847.366} C_VEL
LIN {X 0,Y 559.108,Z 128.835,A -85,B 0,C 180,E1 -2850.149,E2 -2850.149} C_VEL
LIN {X 0,Y 559.16,Z 128.833,A -85,B 0,C 180,E1 -2853.174,E2 -2853.174} C_VEL
LIN {X 0,Y 559.111,Z 128.835,A -85,B 0,C 180,E1 -2855.493,E2 -2855.493} C_VEL
LIN {X 0,Y 559.167,Z 128.836,A -85,B 0,C 180,E1 -2858.624,E2 -2858.624} C_VEL
LIN {X 0,Y 559.15,Z 128.834,A -85,B 0,C 180,E1 -2860.925,E2 -2860.925} C_VEL
LIN {X 0,Y 559.122,Z 128.835,A -85,B 0,C 180,E1 -2863.946,E2 -2863.946} C_VEL
LIN {X 0,Y 559.138,Z 128.836,A -85,B 0,C 180,E1 -2866.183,E2 -2866.183} C_VEL
LIN {X 0,Y 559.186,Z 128.826,A -85,B 0,C 180,E1 -2869.133,E2 -2869.133} C_VEL
LIN {X 0,Y 559.138,Z 128.837,A -85,B 0,C 180,E1 -2872.053,E2 -2872.053} C_VEL
LIN {X 0,Y 559.222,Z 128.821,A -85,B 0,C 180,E1 -2874.953,E2 -2874.953} C_VEL
LIN {X 0,Y 559.245,Z 128.823,A -85,B 0,C 180,E1 -2877.839,E2 -2877.839} C_VEL
LIN {X 0,Y 559.249,Z 128.826,A -85,B 0,C 180,E1 -2880,E2 -2880} C_VEL
LIN {X 0,Y 559.2,Z 128.823,A -85,B 0,C 180,E1 -2882.882,E2 -2882.882} C_VEL
LIN {X 0,Y 559.198,Z 128.831,A -85,B 0,C 180,E1 -2885.77,E2 -2885.77} C_VEL
LIN {X 0,Y 559.144,Z 128.83,A -85,B 0,C 180,E1 -2888.675,E2 -2888.675} C_VEL
LIN {X 0,Y 559.148,Z 128.837,A -85,B 0,C 180,E1 -2891.602,E2 -2891.602} C_VEL
LIN {X 0,Y 559.148,Z 128.83,A -85,B 0,C 180,E1 -2894.576,E2 -2894.576} C_VEL
LIN {X 0,Y 559.106,Z 128.845,A -85,B 0,C 180,E1 -2897.559,E2 -2897.559} C_VEL
LIN {X 0,Y 559.132,Z 128.836,A -85,B 0,C 180,E1 -2899.839,E2 -2899.839} C_VEL
LIN {X 0,Y 559.097,Z 128.837,A -85,B 0,C 180,E1 -2902.155,E2 -2902.155} C_VEL
LIN {X 0,Y 559.134,Z 128.838,A -85,B 0,C 180,E1 -2905.178,E2 -2905.178} C_VEL
LIN {X 0,Y 559.098,Z 128.839,A -85,B 0,C 180,E1 -2907.717,E2 -2907.717} C_VEL
LIN {X 0,Y 559.089,Z 128.837,A -85,B 0,C 180,E1 -2910.187,E2 -2910.187} C_VEL
LIN {X 0,Y 559.143,Z 128.834,A -85,B 0,C 180,E1 -2912.716,E2 -2912.716} C_VEL
LIN {X 0,Y 559.112,Z 128.84,A -85,B 0,C 180,E1 -2915.325,E2 -2915.325} C_VEL
LIN {X 0,Y 559.123,Z 128.833,A -85,B 0,C 180,E1 -2918.019,E2 -2918.019} C_VEL
LIN {X 0,Y 559.15,Z 128.837,A -85,B 0,C 180,E1 -2920.813,E2 -2920.813} C_VEL
LIN {X 0,Y 559.105,Z 128.835,A -85,B 0,C 180,E1 -2923.738,E2 -2923.738} C_VEL
LIN {X 0,Y 559.106,Z 128.837,A -85,B 0,C 180,E1 -2926.263,E2 -2926.263} C_VEL
LIN {X 0,Y 559.151,Z 128.832,A -85,B 0,C 180,E1 -2929.187,E2 -2929.187} C_VEL
LIN {X 0,Y 559.123,Z 128.834,A -85,B 0,C 180,E1 -2931.982,E2 -2931.982} C_VEL
LIN {X 0,Y 559.122,Z 128.838,A -85,B 0,C 180,E1 -2934.789,E2 -2934.789} C_VEL
LIN {X 0,Y 559.149,Z 128.83,A -85,B 0,C 180,E1 -2937.366,E2 -2937.366} C_VEL
LIN {X 0,Y 559.12,Z 128.84,A -85,B 0,C 180,E1 -2940.148,E2 -2940.148} C_VEL
LIN {X 0,Y 559.126,Z 128.835,A -85,B 0,C 180,E1 -2943.182,E2 -2943.182} C_VEL
LIN {X 0,Y 559.158,Z 128.838,A -85,B 0,C 180,E1 -2946.259,E2 -2946.259} C_VEL
LIN {X 0,Y 560.045,Z 134.233,A -85,B 0,C 180,E1 -2947.106,E2 -2947.106} C_VEL
LIN {X 0,Y 559.849,Z 151.334,A -85,B 0,C 180,E1 -2949.613,E2 -2949.613} C_VEL
LIN {X 0,Y 559.582,Z 172.404,A -85,B 0,C 180,E1 -2952.653,E2 -2952.653} C_VEL
LIN {X 0,Y 559.397,Z 193.333,A -85,B 0,C 180,E1 -2955.633,E2 -2955.633} C_VEL
LIN {X 0,Y 559.374,Z 194.479,A -85,B 0,C 180,E1 -2955.795,E2 -2955.795} C_VEL
LIN {X 0,Y 560.255,Z 202.18,A -85,B 0,C 180,E1 -2955.933,E2 -2955.933} C_VEL
LIN {X 0,Y 560.033,Z 302.935,A -85,B 0,C 180,E1 -2957.244,E2 -2957.244} C_VEL
LIN {X 0,Y 559.913,Z 316.21,A -85,B 0,C 180,E1 -2957.564,E2 -2957.564} C_VEL
LIN {X 0,Y 559.792,Z 328.371,A -85,B 0,C 180,E1 -2957.999,E2 -2957.999} C_VEL
LIN {X 0,Y 559.644,Z 340.052,A -85,B 0,C 180,E1 -2958.56,E2 -2958.56} C_VEL
LIN {X 0,Y 559.458,Z 352.19,A -85,B 0,C 180,E1 -2959.322,E2 -2959.322} C_VEL
LIN {X 0,Y 559.305,Z 362.602,A -85,B 0,C 180,E1 -2960.142,E2 -2960.142} C_VEL
LIN {X 0,Y 559.162,Z 371.111,A -85,B 0,C 180,E1 -2960.961,E2 -2960.961} C_VEL
LIN {X 0,Y 559.05,Z 378.958,A -85,B 0,C 180,E1 -2961.869,E2 -2961.869} C_VEL
LIN {X 0,Y 558.944,Z 386.621,A -85,B 0,C 180,E1 -2962.958,E2 -2962.958} C_VEL
LIN {X 0,Y 558.936,Z 393.678,A -85,B 0,C 180,E1 -2964.226,E2 -2964.226} C_VEL
LIN {X 0,Y 558.826,Z 398.372,A -85,B 0,C 180,E1 -2965.311,E2 -2965.311} C_VEL
LIN {X 0,Y 558.836,Z 401.957,A -85,B 0,C 180,E1 -2966.395,E2 -2966.395} C_VEL
LIN {X 0,Y 558.799,Z 403.806,A -85,B 0,C 180,E1 -2967.116,E2 -2967.116} C_VEL
LIN {X 0,Y 558.745,Z 406.182,A -85,B 0,C 180,E1 -2968.558,E2 -2968.558} C_VEL
LIN {X 0,Y 558.74,Z 407,A -85,B 0,C 180,E1 -2970,E2 -2970} C_VEL
LIN {X 0,Y 558.745,Z 406.185,A -85,B 0,C 180,E1 -2971.441,E2 -2971.441} C_VEL
LIN {X 0,Y 558.799,Z 403.811,A -85,B 0,C 180,E1 -2972.883,E2 -2972.883} C_VEL
LIN {X 0,Y 558.844,Z 400.897,A -85,B 0,C 180,E1 -2973.966,E2 -2973.966} C_VEL
LIN {X 0,Y 558.798,Z 396.95,A -85,B 0,C 180,E1 -2975.05,E2 -2975.05} C_VEL
LIN {X 0,Y 558.92,Z 391.87,A -85,B 0,C 180,E1 -2976.135,E2 -2976.135} C_VEL
LIN {X 0,Y 558.977,Z 385.47,A -85,B 0,C 180,E1 -2977.222,E2 -2977.222} C_VEL
LIN {X 0,Y 559.098,Z 377.481,A -85,B 0,C 180,E1 -2978.311,E2 -2978.311} C_VEL
LIN {X 0,Y 559.194,Z 369.338,A -85,B 0,C 180,E1 -2979.22,E2 -2979.22} C_VEL
LIN {X 0,Y 559.357,Z 359.403,A -85,B 0,C 180,E1 -2980.131,E2 -2980.131} C_VEL
LIN {X 0,Y 559.556,Z 348.405,A -85,B 0,C 180,E1 -2980.936,E2 -2980.936} C_VEL
LIN {X 0,Y 559.67,Z 336.467,A -85,B 0,C 180,E1 -2981.627,E2 -2981.627} C_VEL
LIN {X 0,Y 559.821,Z 324.99,A -85,B 0,C 180,E1 -2982.138,E2 -2982.138} C_VEL
LIN {X 0,Y 559.979,Z 312.195,A -85,B 0,C 180,E1 -2982.549,E2 -2982.549} C_VEL
LIN {X 0,Y 560.08,Z 298.631,A -85,B 0,C 180,E1 -2982.823,E2 -2982.823} C_VEL
LIN {X 0,Y 560.2,Z 200.223,A -85,B 0,C 180,E1 -2984.093,E2 -2984.093} C_VEL
LIN {X 0,Y 559.371,Z 194.483,A -85,B 0,C 180,E1 -2984.204,E2 -2984.204} C_VEL
LIN {X 0,Y 559.564,Z 174.367,A -85,B 0,C 180,E1 -2987.066,E2 -2987.066} C_VEL
LIN {X 0,Y 559.831,Z 153.969,A -85,B 0,C 180,E1 -2990.004,E2 -2990.004} C_VEL
LIN {X 0,Y 560.051,Z 135.555,A -85,B 0,C 180,E1 -2992.697,E2 -2992.697} C_VEL
LIN {X 0,Y 559.167,Z 128.941,A -85,B 0,C 180,E1 -2993.715,E2 -2993.715} C_VEL
LIN {X 0,Y 559.139,Z 128.833,A -85,B 0,C 180,E1 -2996.82,E2 -2996.82} C_VEL
LIN {X 0,Y 559.117,Z 128.841,A -85,B 0,C 180,E1 -2999.851,E2 -2999.851} C_VEL
LIN {X 0,Y 559.145,Z 128.83,A -85,B 0,C 180,E1 -3002.715,E2 -3002.715} C_VEL
LIN {X 0,Y 559.113,Z 128.841,A -85,B 0,C 180,E1 -3005.324,E2 -3005.324} C_VEL
LIN {X 0,Y 559.122,Z 128.834,A -85,B 0,C 180,E1 -3008.017,E2 -3008.017} C_VEL
LIN {X 0,Y 559.148,Z 128.832,A -85,B 0,C 180,E1 -3010.812,E2 -3010.812} C_VEL
LIN {X 0,Y 559.129,Z 128.835,A -85,B 0,C 180,E1 -3013.734,E2 -3013.734} C_VEL
LIN {X 0,Y 559.118,Z 128.837,A -85,B 0,C 180,E1 -3016.805,E2 -3016.805} C_VEL
LIN {X 0,Y 559.145,Z 128.838,A -85,B 0,C 180,E1 -3019.186,E2 -3019.186} C_VEL
LIN {X 0,Y 559.119,Z 128.833,A -85,B 0,C 180,E1 -3021.981,E2 -3021.981} C_VEL
LIN {X 0,Y 559.113,Z 128.841,A -85,B 0,C 180,E1 -3024.788,E2 -3024.788} C_VEL
LIN {X 0,Y 559.139,Z 128.833,A -85,B 0,C 180,E1 -3027.365,E2 -3027.365} C_VEL
LIN {X 0,Y 559.101,Z 128.837,A -85,B 0,C 180,E1 -3030.149,E2 -3030.149} C_VEL
LIN {X 0,Y 559.116,Z 128.837,A -85,B 0,C 180,E1 -3033.181,E2 -3033.181} C_VEL
LIN {X 0,Y 559.103,Z 128.835,A -85,B 0,C 180,E1 -3035.492,E2 -3035.492} C_VEL
LIN {X 0,Y 559.148,Z 128.838,A -85,B 0,C 180,E1 -3038.623,E2 -3038.623} C_VEL
LIN {X 0,Y 559.142,Z 128.834,A -85,B 0,C 180,E1 -3040.925,E2 -3040.925} C_VEL
LIN {X 0,Y 559.113,Z 128.837,A -85,B 0,C 180,E1 -3043.946,E2 -3043.946} C_VEL
LIN {X 0,Y 559.129,Z 128.839,A -85,B 0,C 180,E1 -3046.183,E2 -3046.183} C_VEL
LIN {X 0,Y 559.156,Z 128.829,A -85,B 0,C 180,E1 -3049.133,E2 -3049.133} C_VEL
LIN {X 0,Y 559.128,Z 128.84,A -85,B 0,C 180,E1 -3052.053,E2 -3052.053} C_VEL
LIN {X 0,Y 559.215,Z 128.822,A -85,B 0,C 180,E1 -3054.953,E2 -3054.953} C_VEL
LIN {X 0,Y 559.24,Z 128.825,A -85,B 0,C 180,E1 -3057.839,E2 -3057.839} C_VEL
LIN {X 0,Y 559.243,Z 128.827,A -85,B 0,C 180,E1 -3060,E2 -3060} C_VEL
LIN {X 0,Y 559.196,Z 128.824,A -85,B 0,C 180,E1 -3062.882,E2 -3062.882} C_VEL
LIN {X 0,Y 559.204,Z 128.832,A -85,B 0,C 180,E1 -3065.77,E2 -3065.77} C_VEL
LIN {X 0,Y 559.148,Z 128.83,A -85,B 0,C 180,E1 -3068.675,E2 -3068.675} C_VEL
LIN {X 0,Y 559.186,Z 128.834,A -85,B 0,C 180,E1 -3071.601,E2 -3071.601} C_VEL
LIN {X 0,Y 559.149,Z 128.83,A -85,B 0,C 180,E1 -3074.58,E2 -3074.58} C_VEL
LIN {X 0,Y 559.099,Z 128.844,A -85,B 0,C 180,E1 -3077.559,E2 -3077.559} C_VEL
LIN {X 0,Y 559.151,Z 128.833,A -85,B 0,C 180,E1 -3079.838,E2 -3079.838} C_VEL
LIN {X 0,Y 559.121,Z 128.833,A -85,B 0,C 180,E1 -3082.154,E2 -3082.154} C_VEL
LIN {X 0,Y 559.129,Z 128.84,A -85,B 0,C 180,E1 -3085.178,E2 -3085.178} C_VEL
LIN {X 0,Y 559.1,Z 128.838,A -85,B 0,C 180,E1 -3087.717,E2 -3087.717} C_VEL
LIN {X 0,Y 559.118,Z 128.836,A -85,B 0,C 180,E1 -3090.577,E2 -3090.577} C_VEL
LIN {X 0,Y 558.46,Z 128.924,A -85,B 0,C 180,E1 -3091.179,E2 -3091.179} C_VEL
LIN {X 0,Y 555.601,Z 129.28,A -85,B 0,C 180,E1 -3092.155,E2 -3092.155} C_VEL
LIN {X 0,Y 553.185,Z 129.58,A -85,B 0,C 180,E1 -3092.94,E2 -3092.94} C_VEL
LIN {X 0,Y 552.157,Z 129.703,A -85,B 0,C 180,E1 -3093.547,E2 -3093.547} C_VEL
LIN {X 0,Y 552.078,Z 129.711,A -85,B 0,C 180,E1 -3093.752,E2 -3093.752} C_VEL
LIN {X 0,Y 552.098,Z 129.714,A -85,B 0,C 180,E1 -3096.748,E2 -3096.748} C_VEL
LIN {X 0,Y 552.119,Z 129.706,A -85,B 0,C 180,E1 -3099.528,E2 -3099.528} C_VEL
LIN {X 0,Y 552.101,Z 129.712,A -85,B 0,C 180,E1 -3102.429,E2 -3102.429} C_VEL
LIN {X 0,Y 552.086,Z 129.71,A -85,B 0,C 180,E1 -3105.563,E2 -3105.563} C_VEL
LIN {X 0,Y 552.103,Z 129.716,A -85,B 0,C 180,E1 -3108.681,E2 -3108.681} C_VEL
LIN {X 0,Y 552.109,Z 129.707,A -85,B 0,C 180,E1 -3111.412,E2 -3111.412} C_VEL
LIN {X 0,Y 552.071,Z 129.716,A -85,B 0,C 180,E1 -3114.156,E2 -3114.156} C_VEL
LIN {X 0,Y 552.11,Z 129.71,A -85,B 0,C 180,E1 -3116.815,E2 -3116.815} C_VEL
LIN {X 0,Y 552.091,Z 129.709,A -85,B 0,C 180,E1 -3119.391,E2 -3119.391} C_VEL
LIN {X 0,Y 552.066,Z 129.716,A -85,B 0,C 180,E1 -3121.9,E2 -3121.9} C_VEL
LIN {X 0,Y 552.085,Z 129.712,A -85,B 0,C 180,E1 -3124.666,E2 -3124.666} C_VEL
LIN {X 0,Y 552.086,Z 129.712,A -85,B 0,C 180,E1 -3127.55,E2 -3127.55} C_VEL
LIN {X 0,Y 552.171,Z 129.706,A -85,B 0,C 180,E1 -3130.624,E2 -3130.624} C_VEL
LIN {X 0,Y 552.269,Z 130.752,A -85,B 0,C 180,E1 -3130.872,E2 -3130.872} C_VEL
LIN {X 0,Y 552.433,Z 137.979,A -85,B 0,C 180,E1 -3132.223,E2 -3132.223} C_VEL
LIN {X 0,Y 552.287,Z 153.404,A -85,B 0,C 180,E1 -3135.068,E2 -3135.068} C_VEL
LIN {X 0,Y 552.236,Z 156.793,A -85,B 0,C 180,E1 -3135.69,E2 -3135.69} C_VEL
LIN {X 0,Y 553.441,Z 164.702,A -85,B 0,C 180,E1 -3135.827,E2 -3135.827} C_VEL
LIN {X 0,Y 553.142,Z 263.424,A -85,B 0,C 180,E1 -3137.13,E2 -3137.13} C_VEL
LIN {X 0,Y 552.973,Z 276.63,A -85,B 0,C 180,E1 -3137.453,E2 -3137.453} C_VEL
LIN {X 0,Y 552.841,Z 288.745,A -85,B 0,C 180,E1 -3137.893,E2 -3137.893} C_VEL
LIN {X 0,Y 552.709,Z 300.207,A -85,B 0,C 180,E1 -3138.452,E2 -3138.452} C_VEL
LIN {X 0,Y 552.495,Z 311.824,A -85,B 0,C 180,E1 -3139.186,E2 -3139.186} C_VEL
LIN {X 0,Y 552.304,Z 322.294,A -85,B 0,C 180,E1 -3140.016,E2 -3140.016} C_VEL
LIN {X 0,Y 552.178,Z 330.846,A -85,B 0,C 180,E1 -3140.846,E2 -3140.846} C_VEL
LIN {X 0,Y 552.007,Z 338.723,A -85,B 0,C 180,E1 -3141.766,E2 -3141.766} C_VEL
LIN {X 0,Y 551.916,Z 346.534,A -85,B 0,C 180,E1 -3142.887,E2 -3142.887} C_VEL
LIN {X 0,Y 551.868,Z 353.482,A -85,B 0,C 180,E1 -3144.153,E2 -3144.153} C_VEL
LIN {X 0,Y 551.725,Z 358.198,A -85,B 0,C 180,E1 -3145.251,E2 -3145.251} C_VEL
LIN {X 0,Y 551.75,Z 361.83,A -85,B 0,C 180,E1 -3146.349,E2 -3146.349} C_VEL
LIN {X 0,Y 551.723,Z 363.708,A -85,B 0,C 180,E1 -3147.08,E2 -3147.08} C_VEL
LIN {X 0,Y 551.657,Z 365.127,A -85,B 0,C 180,E1 -3147.81,E2 -3147.81} C_VEL
LIN {X 0,Y 551.642,Z 366.756,A -85,B 0,C 180,E1 -3149.27,E2 -3149.27} C_VEL
LIN {X 0,Y 551.641,Z 366.996,A -85,B 0,C 180,E1 -3150,E2 -3150} C_VEL
LIN {X 0,Y 551.641,Z 366.815,A -85,B 0,C 180,E1 -3150.73,E2 -3150.73} C_VEL
LIN {X 0,Y 551.657,Z 365.261,A -85,B 0,C 180,E1 -3152.191,E2 -3152.191} C_VEL
LIN {X 0,Y 551.724,Z 363.901,A -85,B 0,C 180,E1 -3152.921,E2 -3152.921} C_VEL
LIN {X 0,Y 551.764,Z 361.024,A -85,B 0,C 180,E1 -3154.017,E2 -3154.017} C_VEL
LIN {X 0,Y 551.723,Z 357.125,A -85,B 0,C 180,E1 -3155.116,E2 -3155.116} C_VEL
LIN {X 0,Y 551.834,Z 351.431,A -85,B 0,C 180,E1 -3156.349,E2 -3156.349} C_VEL
LIN {X 0,Y 551.926,Z 344.617,A -85,B 0,C 180,E1 -3157.5,E2 -3157.5} C_VEL
LIN {X 0,Y 552.063,Z 336.484,A -85,B 0,C 180,E1 -3158.603,E2 -3158.603} C_VEL
LIN {X 0,Y 552.221,Z 328.158,A -85,B 0,C 180,E1 -3159.524,E2 -3159.524} C_VEL
LIN {X 0,Y 552.414,Z 319.044,A -85,B 0,C 180,E1 -3160.353,E2 -3160.353} C_VEL
LIN {X 0,Y 552.563,Z 308.312,A -85,B 0,C 180,E1 -3161.144,E2 -3161.144} C_VEL
LIN {X 0,Y 552.778,Z 296.557,A -85,B 0,C 180,E1 -3161.83,E2 -3161.83} C_VEL
LIN {X 0,Y 552.928,Z 284.059,A -85,B 0,C 180,E1 -3162.386,E2 -3162.386} C_VEL
LIN {X 0,Y 553.1,Z 270.637,A -85,B 0,C 180,E1 -3162.801,E2 -3162.801} C_VEL
LIN {X 0,Y 553.196,Z 258.85,A -85,B 0,C 180,E1 -3163.033,E2 -3163.033} C_VEL
LIN {X 0,Y 553.356,Z 163.113,A -85,B 0,C 180,E1 -3164.286,E2 -3164.286} C_VEL
LIN {X 0,Y 552.198,Z 156.766,A -85,B 0,C 180,E1 -3164.407,E2 -3164.407} C_VEL
LIN {X 0,Y 552.39,Z 141.123,A -85,B 0,C 180,E1 -3167.286,E2 -3167.286} C_VEL
LIN {X 0,Y 552.363,Z 131.23,A -85,B 0,C 180,E1 -3169.125,E2 -3169.125} C_VEL
LIN {X 0,Y 552.154,Z 129.709,A -85,B 0,C 180,E1 -3169.429,E2 -3169.429} C_VEL
LIN {X 0,Y 552.089,Z 129.712,A -85,B 0,C 180,E1 -3172.451,E2 -3172.451} C_VEL
LIN {X 0,Y 552.088,Z 129.711,A -85,B 0,C 180,E1 -3175.335,E2 -3175.335} C_VEL
LIN {X 0,Y 552.079,Z 129.716,A -85,B 0,C 180,E1 -3178.1,E2 -3178.1} C_VEL
LIN {X 0,Y 552.094,Z 129.709,A -85,B 0,C 180,E1 -3180.61,E2 -3180.61} C_VEL
LIN {X 0,Y 552.114,Z 129.708,A -85,B 0,C 180,E1 -3183.186,E2 -3183.186} C_VEL
LIN {X 0,Y 552.075,Z 129.717,A -85,B 0,C 180,E1 -3185.844,E2 -3185.844} C_VEL
LIN {X 0,Y 552.114,Z 129.706,A -85,B 0,C 180,E1 -3188.589,E2 -3188.589} C_VEL
LIN {X 0,Y 552.11,Z 129.716,A -85,B 0,C 180,E1 -3191.447,E2 -3191.447} C_VEL
LIN {X 0,Y 552.088,Z 129.709,A -85,B 0,C 180,E1 -3194.531,E2 -3194.531} C_VEL
LIN {X 0,Y 552.108,Z 129.712,A -85,B 0,C 180,E1 -3197.587,E2 -3197.587} C_VEL
LIN {X 0,Y 552.124,Z 129.705,A -85,B 0,C 180,E1 -3200.472,E2 -3200.472} C_VEL
LIN {X 0,Y 552.097,Z 129.715,A -85,B 0,C 180,E1 -3203.318,E2 -3203.318} C_VEL
LIN {X 0,Y 552.096,Z 129.708,A -85,B 0,C 180,E1 -3205.937,E2 -3205.937} C_VEL
LIN {X 0,Y 552.101,Z 129.711,A -85,B 0,C 180,E1 -3208.539,E2 -3208.539} C_VEL
LIN {X 0,Y 552.076,Z 129.713,A -85,B 0,C 180,E1 -3211.447,E2 -3211.447} C_VEL
LIN {X 0,Y 552.107,Z 129.708,A -85,B 0,C 180,E1 -3213.543,E2 -3213.543} C_VEL
LIN {X 0,Y 552.085,Z 129.719,A -85,B 0,C 180,E1 -3216.757,E2 -3216.757} C_VEL
LIN {X 0,Y 552.11,Z 129.709,A -85,B 0,C 180,E1 -3219.119,E2 -3219.119} C_VEL
LIN {X 0,Y 552.075,Z 129.711,A -85,B 0,C 180,E1 -3221.443,E2 -3221.443} C_VEL
LIN {X 0,Y 552.082,Z 129.719,A -85,B 0,C 180,E1 -3224.494,E2 -3224.494} C_VEL
LIN {X 0,Y 552.095,Z 129.713,A -85,B 0,C 180,E1 -3226.754,E2 -3226.754} C_VEL
LIN {X 0,Y 552.155,Z 129.702,A -85,B 0,C 180,E1 -3228.993,E2 -3228.993} C_VEL
LIN {X 0,Y 552.106,Z 129.711,A -85,B 0,C 180,E1 -3231.951,E2 -3231.951} C_VEL
LIN {X 0,Y 552.199,Z 129.696,A -85,B 0,C 180,E1 -3234.889,E2 -3234.889} C_VEL
LIN {X 0,Y 552.215,Z 129.698,A -85,B 0,C 180,E1 -3237.812,E2 -3237.812} C_VEL
LIN {X 0,Y 552.217,Z 129.701,A -85,B 0,C 180,E1 -3240,E2 -3240} C_VEL
LIN {X 0,Y 552.168,Z 129.699,A -85,B 0,C 180,E1 -3242.918,E2 -3242.918} C_VEL
LIN {X 0,Y 552.168,Z 129.708,A -85,B 0,C 180,E1 -3245.844,E2 -3245.844} C_VEL
LIN {X 0,Y 552.117,Z 129.706,A -85,B 0,C 180,E1 -3248.786,E2 -3248.786} C_VEL
LIN {X 0,Y 552.092,Z 129.718,A -85,B 0,C 180,E1 -3251.752,E2 -3251.752} C_VEL
LIN {X 0,Y 552.085,Z 129.71,A -85,B 0,C 180,E1 -3254.75,E2 -3254.75} C_VEL
LIN {X 0,Y 552.069,Z 129.718,A -85,B 0,C 180,E1 -3257.79,E2 -3257.79} C_VEL
LIN {X 0,Y 552.087,Z 129.711,A -85,B 0,C 180,E1 -3260.103,E2 -3260.103} C_VEL
LIN {X 0,Y 552.037,Z 129.715,A -85,B 0,C 180,E1 -3262.453,E2 -3262.453} C_VEL
LIN {X 0,Y 552.076,Z 129.72,A -85,B 0,C 180,E1 -3265.334,E2 -3265.334} C_VEL
LIN {X 0,Y 552.045,Z 129.715,A -85,B 0,C 180,E1 -3268.102,E2 -3268.102} C_VEL
LIN {X 0,Y 552.065,Z 129.714,A -85,B 0,C 180,E1 -3270.612,E2 -3270.612} C_VEL
LIN {X 0,Y 552.1,Z 129.717,A -85,B 0,C 180,E1 -3273.187,E2 -3273.187} C_VEL
LIN {X 0,Y 552.067,Z 129.712,A -85,B 0,C 180,E1 -3275.845,E2 -3275.845} C_VEL
LIN {X 0,Y 552.11,Z 129.71,A -85,B 0,C 180,E1 -3278.59,E2 -3278.59} C_VEL
LIN {X 0,Y 552.071,Z 129.713,A -85,B 0,C 180,E1 -3281.451,E2 -3281.451} C_VEL
LIN {X 0,Y 552.073,Z 129.716,A -85,B 0,C 180,E1 -3284.53,E2 -3284.53} C_VEL
LIN {X 0,Y 552.085,Z 129.71,A -85,B 0,C 180,E1 -3287.59,E2 -3287.59} C_VEL
LIN {X 0,Y 552.124,Z 129.712,A -85,B 0,C 180,E1 -3290.472,E2 -3290.472} C_VEL
LIN {X 0,Y 552.097,Z 129.709,A -85,B 0,C 180,E1 -3293.319,E2 -3293.319} C_VEL
LIN {X 0,Y 552.097,Z 129.71,A -85,B 0,C 180,E1 -3295.937,E2 -3295.937} C_VEL
LIN {X 0,Y 552.121,Z 129.713,A -85,B 0,C 180,E1 -3298.541,E2 -3298.541} C_VEL
LIN {X 0,Y 552.084,Z 129.711,A -85,B 0,C 180,E1 -3301.446,E2 -3301.446} C_VEL
LIN {X 0,Y 552.085,Z 129.719,A -85,B 0,C 180,E1 -3304.354,E2 -3304.354} C_VEL
LIN {X 0,Y 552.099,Z 129.818,A -85,B 0,C 180,E1 -3306.133,E2 -3306.133} C_VEL
LIN {X 0,Y 553.064,Z 135.306,A -85,B 0,C 180,E1 -3306.999,E2 -3306.999} C_VEL
LIN {X 0,Y 552.946,Z 148.459,A -85,B 0,C 180,E1 -3308.957,E2 -3308.957} C_VEL
LIN {X 0,Y 552.682,Z 168.16,A -85,B 0,C 180,E1 -3311.847,E2 -3311.847} C_VEL
LIN {X 0,Y 552.395,Z 187.829,A -85,B 0,C 180,E1 -3314.692,E2 -3314.692} C_VEL
LIN {X 0,Y 552.362,Z 194.334,A -85,B 0,C 180,E1 -3315.627,E2 -3315.627} C_VEL
LIN {X 0,Y 553.36,Z 202.461,A -85,B 0,C 180,E1 -3315.762,E2 -3315.762} C_VEL
LIN {X 0,Y 553.116,Z 302.676,A -85,B 0,C 180,E1 -3317.082,E2 -3317.082} C_VEL
LIN {X 0,Y 552.98,Z 315.971,A -85,B 0,C 180,E1 -3317.406,E2 -3317.406} C_VEL
LIN {X 0,Y 552.847,Z 328.154,A -85,B 0,C 180,E1 -3317.845,E2 -3317.845} C_VEL
LIN {X 0,Y 552.657,Z 338.979,A -85,B 0,C 180,E1 -3318.365,E2 -3318.365} C_VEL
LIN {X 0,Y 552.482,Z 350.767,A -85,B 0,C 180,E1 -3319.092,E2 -3319.092} C_VEL
LIN {X 0,Y 552.298,Z 361.45,A -85,B 0,C 180,E1 -3319.923,E2 -3319.923} C_VEL
LIN {X 0,Y 552.131,Z 371.077,A -85,B 0,C 180,E1 -3320.844,E2 -3320.844} C_VEL
LIN {X 0,Y 552.013,Z 378.958,A -85,B 0,C 180,E1 -3321.765,E2 -3321.765} C_VEL
LIN {X 0,Y 551.89,Z 386.619,A -85,B 0,C 180,E1 -3322.867,E2 -3322.867} C_VEL
LIN {X 0,Y 551.867,Z 393.678,A -85,B 0,C 180,E1 -3324.152,E2 -3324.152} C_VEL
LIN {X 0,Y 551.725,Z 398.372,A -85,B 0,C 180,E1 -3325.25,E2 -3325.25} C_VEL
LIN {X 0,Y 551.75,Z 401.957,A -85,B 0,C 180,E1 -3326.348,E2 -3326.348} C_VEL
LIN {X 0,Y 551.723,Z 403.806,A -85,B 0,C 180,E1 -3327.079,E2 -3327.079} C_VEL
LIN {X 0,Y 551.645,Z 406.181,A -85,B 0,C 180,E1 -3328.54,E2 -3328.54} C_VEL
LIN {X 0,Y 551.64,Z 407,A -85,B 0,C 180,E1 -3330,E2 -3330} C_VEL
LIN {X 0,Y 551.645,Z 406.184,A -85,B 0,C 180,E1 -3331.46,E2 -3331.46} C_VEL
LIN {X 0,Y 551.723,Z 403.811,A -85,B 0,C 180,E1 -3332.92,E2 -3332.92} C_VEL
LIN {X 0,Y 551.764,Z 400.896,A -85,B 0,C 180,E1 -3334.017,E2 -3334.017} C_VEL
LIN {X 0,Y 551.723,Z 396.95,A -85,B 0,C 180,E1 -3335.115,E2 -3335.115} C_VEL
LIN {X 0,Y 551.823,Z 391.196,A -85,B 0,C 180,E1 -3336.34,E2 -3336.34} C_VEL
LIN {X 0,Y 551.926,Z 384.238,A -85,B 0,C 180,E1 -3337.499,E2 -3337.499} C_VEL
LIN {X 0,Y 552.082,Z 375.991,A -85,B 0,C 180,E1 -3338.602,E2 -3338.602} C_VEL
LIN {X 0,Y 552.2,Z 367.493,A -85,B 0,C 180,E1 -3339.523,E2 -3339.523} C_VEL
LIN {X 0,Y 552.428,Z 356.995,A -85,B 0,C 180,E1 -3340.444,E2 -3340.444} C_VEL
LIN {X 0,Y 552.574,Z 346.145,A -85,B 0,C 180,E1 -3341.214,E2 -3341.214} C_VEL
LIN {X 0,Y 552.751,Z 335.227,A -85,B 0,C 180,E1 -3341.83,E2 -3341.83} C_VEL
LIN {X 0,Y 552.897,Z 323.558,A -85,B 0,C 180,E1 -3342.339,E2 -3342.339} C_VEL
LIN {X 0,Y 553.039,Z 311.033,A -85,B 0,C 180,E1 -3342.732,E2 -3342.732} C_VEL
LIN {X 0,Y 553.169,Z 298.372,A -85,B 0,C 180,E1 -3342.986,E2 -3342.986} C_VEL
LIN {X 0,Y 553.231,Z 200.445,A -85,B 0,C 180,E1 -3344.268,E2 -3344.268} C_VEL
LIN {X 0,Y 552.366,Z 194.199,A -85,B 0,C 180,E1 -3344.392,E2 -3344.392} C_VEL
LIN {X 0,Y 552.566,Z 173.728,A -85,B 0,C 180,E1 -3347.344,E2 -3347.344} C_VEL
LIN {X 0,Y 552.895,Z 153.721,A -85,B 0,C 180,E1 -3350.265,E2 -3350.265} C_VEL
LIN {X 0,Y 553.104,Z 136.63,A -85,B 0,C 180,E1 -3352.801,E2 -3352.801} C_VEL
LIN {X 0,Y 552.401,Z 131.196,A -85,B 0,C 180,E1 -3353.647,E2 -3353.647} C_VEL
LIN {X 0,Y 552.086,Z 129.719,A -85,B 0,C 180,E1 -3353.914,E2 -3353.914} C_VEL
LIN {X 0,Y 552.093,Z 129.711,A -85,B 0,C 180,E1 -3356.457,E2 -3356.457} C_VEL
LIN {X 0,Y 552.052,Z 129.716,A -85,B 0,C 180,E1 -3358.931,E2 -3358.931} C_VEL
LIN {X 0,Y 552.109,Z 129.715,A -85,B 0,C 180,E1 -3361.475,E2 -3361.475} C_VEL
LIN {X 0,Y 552.093,Z 129.71,A -85,B 0,C 180,E1 -3364.164,E2 -3364.164} C_VEL
LIN {X 0,Y 552.093,Z 129.709,A -85,B 0,C 180,E1 -3366.747,E2 -3366.747} C_VEL
LIN {X 0,Y 552.121,Z 129.712,A -85,B 0,C 180,E1 -3369.527,E2 -3369.527} C_VEL
LIN {X 0,Y 552.102,Z 129.708,A -85,B 0,C 180,E1 -3372.427,E2 -3372.427} C_VEL
LIN {X 0,Y 552.068,Z 129.716,A -85,B 0,C 180,E1 -3375.559,E2 -3375.559} C_VEL
LIN {X 0,Y 552.069,Z 129.715,A -85,B 0,C 180,E1 -3378.683,E2 -3378.683} C_VEL
LIN {X 0,Y 552.105,Z 129.711,A -85,B 0,C 180,E1 -3381.41,E2 -3381.41} C_VEL
LIN {X 0,Y 552.062,Z 129.713,A -85,B 0,C 180,E1 -3384.154,E2 -3384.154} C_VEL
LIN {X 0,Y 552.097,Z 129.713,A -85,B 0,C 180,E1 -3387.155,E2 -3387.155} C_VEL
LIN {X 0,Y 552.079,Z 129.711,A -85,B 0,C 180,E1 -3389.954,E2 -3389.954} C_VEL
LIN {X 0,Y 552.083,Z 129.715,A -85,B 0,C 180,E1 -3393.009,E2 -3393.009} C_VEL
LIN {X 0,Y 552.066,Z 129.713,A -85,B 0,C 180,E1 -3395.96,E2 -3395.96} C_VEL
LIN {X 0,Y 552.085,Z 129.711,A -85,B 0,C 180,E1 -3399.118,E2 -3399.118} C_VEL
LIN {X 0,Y 552.066,Z 129.712,A -85,B 0,C 180,E1 -3401.442,E2 -3401.442} C_VEL
LIN {X 0,Y 552.073,Z 129.719,A -85,B 0,C 180,E1 -3404.494,E2 -3404.494} C_VEL
LIN {X 0,Y 552.086,Z 129.713,A -85,B 0,C 180,E1 -3406.754,E2 -3406.754} C_VEL
LIN {X 0,Y 552.075,Z 129.713,A -85,B 0,C 180,E1 -3409.734,E2 -3409.734} C_VEL
LIN {X 0,Y 552.096,Z 129.714,A -85,B 0,C 180,E1 -3411.951,E2 -3411.951} C_VEL
LIN {X 0,Y 552.192,Z 129.697,A -85,B 0,C 180,E1 -3414.889,E2 -3414.889} C_VEL
LIN {X 0,Y 552.21,Z 129.7,A -85,B 0,C 180,E1 -3417.812,E2 -3417.812} C_VEL
LIN {X 0,Y 552.212,Z 129.703,A -85,B 0,C 180,E1 -3420,E2 -3420} C_VEL
LIN {X 0,Y 552.165,Z 129.7,A -85,B 0,C 180,E1 -3422.918,E2 -3422.918} C_VEL
LIN {X 0,Y 552.173,Z 129.708,A -85,B 0,C 180,E1 -3425.844,E2 -3425.844} C_VEL
LIN {X 0,Y 552.12,Z 129.705,A -85,B 0,C 180,E1 -3428.786,E2 -3428.786} C_VEL
LIN {X 0,Y 552.141,Z 129.71,A -85,B 0,C 180,E1 -3431.751,E2 -3431.751} C_VEL
LIN {X 0,Y 552.11,Z 129.707,A -85,B 0,C 180,E1 -3434.749,E2 -3434.749} C_VEL
LIN {X 0,Y 552.065,Z 129.717,A -85,B 0,C 180,E1 -3437.79,E2 -3437.79} C_VEL
LIN {X 0,Y 552.112,Z 129.707,A -85,B 0,C 180,E1 -3440.102,E2 -3440.102} C_VEL
LIN {X 0,Y 552.073,Z 129.711,A -85,B 0,C 180,E1 -3442.452,E2 -3442.452} C_VEL
LIN {X 0,Y 552.073,Z 129.719,A -85,B 0,C 180,E1 -3445.335,E2 -3445.335} C_VEL
LIN {X 0,Y 552.048,Z 129.714,A -85,B 0,C 180,E1 -3448.102,E2 -3448.102} C_VEL
LIN {X 0,Y 552.083,Z 129.712,A -85,B 0,C 180,E1 -3450.611,E2 -3450.611} C_VEL
LIN {X 0,Y 552.096,Z 129.715,A -85,B 0,C 180,E1 -3453.187,E2 -3453.187} C_VEL
LIN {X 0,Y 552.078,Z 129.711,A -85,B 0,C 180,E1 -3453.752,E2 -3453.752} C_VEL
LIN {X 0,Y 551.438,Z 129.792,A -85,B 0,C 180,E1 -3454.361,E2 -3454.361} C_VEL
LIN {X 0,Y 548.629,Z 130.151,A -85,B 0,C 180,E1 -3455.35,E2 -3455.35} C_VEL
LIN {X 0,Y 546.224,Z 130.455,A -85,B 0,C 180,E1 -3456.145,E2 -3456.145} C_VEL
LIN {X 0,Y 545.16,Z 130.584,A -85,B 0,C 180,E1 -3456.759,E2 -3456.759} C_VEL
LIN {X 0,Y 545.057,Z 130.594,A -85,B 0,C 180,E1 -3456.967,E2 -3456.967} C_VEL
LIN {X 0,Y 545.056,Z 130.586,A -85,B 0,C 180,E1 -3460.144,E2 -3460.144} C_VEL
LIN {X 0,Y 545.016,Z 130.594,A -85,B 0,C 180,E1 -3463.113,E2 -3463.113} C_VEL
LIN {X 0,Y 545.044,Z 130.59,A -85,B 0,C 180,E1 -3466.227,E2 -3466.227} C_VEL
LIN {X 0,Y 545.067,Z 130.589,A -85,B 0,C 180,E1 -3468.885,E2 -3468.885} C_VEL
LIN {X 0,Y 545.073,Z 130.588,A -85,B 0,C 180,E1 -3470.819,E2 -3470.819} C_VEL
LIN {X 0,Y 545.03,Z 130.589,A -85,B 0,C 180,E1 -3473.62,E2 -3473.62} C_VEL
LIN {X 0,Y 545.061,Z 130.593,A -85,B 0,C 180,E1 -3476.329,E2 -3476.329} C_VEL
LIN {X 0,Y 545.06,Z 130.586,A -85,B 0,C 180,E1 -3478.953,E2 -3478.953} C_VEL
LIN {X 0,Y 545.043,Z 130.587,A -85,B 0,C 180,E1 -3481.505,E2 -3481.505} C_VEL
LIN {X 0,Y 545.048,Z 130.591,A -85,B 0,C 180,E1 -3484.502,E2 -3484.502} C_VEL
LIN {X 0,Y 545.031,Z 130.589,A -85,B 0,C 180,E1 -3487.243,E2 -3487.243} C_VEL
LIN {X 0,Y 545.12,Z 130.586,A -85,B 0,C 180,E1 -3490.416,E2 -3490.416} C_VEL
LIN {X 0,Y 545.152,Z 130.79,A -85,B 0,C 180,E1 -3490.613,E2 -3490.613} C_VEL
LIN {X 0,Y 545.495,Z 135.963,A -85,B 0,C 180,E1 -3491.601,E2 -3491.601} C_VEL
LIN {X 0,Y 545.272,Z 152.517,A -85,B 0,C 180,E1 -3494.68,E2 -3494.68} C_VEL
LIN {X 0,Y 545.216,Z 156.975,A -85,B 0,C 180,E1 -3495.5,E2 -3495.5} C_VEL
LIN {X 0,Y 546.534,Z 164.411,A -85,B 0,C 180,E1 -3495.636,E2 -3495.636} C_VEL
LIN {X 0,Y 546.234,Z 263.712,A -85,B 0,C 180,E1 -3496.965,E2 -3496.965} C_VEL
LIN {X 0,Y 546.071,Z 276.908,A -85,B 0,C 180,E1 -3497.292,E2 -3497.292} C_VEL
LIN {X 0,Y 545.933,Z 289.009,A -85,B 0,C 180,E1 -3497.737,E2 -3497.737} C_VEL
LIN {X 0,Y 545.75,Z 301.151,A -85,B 0,C 180,E1 -3498.342,E2 -3498.342} C_VEL
LIN {X 0,Y 545.546,Z 312.09,A -85,B 0,C 180,E1 -3499.047,E2 -3499.047} C_VEL
LIN {X 0,Y 545.322,Z 322.56,A -85,B 0,C 180,E1 -3499.887,E2 -3499.887} C_VEL
LIN {X 0,Y 545.17,Z 331.111,A -85,B 0,C 180,E1 -3500.727,E2 -3500.727} C_VEL
LIN {X 0,Y 544.975,Z 338.987,A -85,B 0,C 180,E1 -3501.659,E2 -3501.659} C_VEL
LIN {X 0,Y 544.867,Z 346.686,A -85,B 0,C 180,E1 -3502.776,E2 -3502.776} C_VEL
LIN {X 0,Y 544.801,Z 353.744,A -85,B 0,C 180,E1 -3504.077,E2 -3504.077} C_VEL
LIN {X 0,Y 544.654,Z 358.453,A -85,B 0,C 180,E1 -3505.189,E2 -3505.189} C_VEL
LIN {X 0,Y 544.669,Z 362.055,A -85,B 0,C 180,E1 -3506.301,E2 -3506.301} C_VEL
LIN {X 0,Y 544.65,Z 363.918,A -85,B 0,C 180,E1 -3507.042,E2 -3507.042} C_VEL
LIN {X 0,Y 544.572,Z 365.328,A -85,B 0,C 180,E1 -3507.782,E2 -3507.782} C_VEL
LIN {X 0,Y 544.545,Z 366.944,A -85,B 0,C 180,E1 -3509.261,E2 -3509.261} C_VEL
LIN {X 0,Y 544.544,Z 367.182,A -85,B 0,C 180,E1 -3510,E2 -3510} C_VEL
LIN {X 0,Y 544.544,Z 367.001,A -85,B 0,C 180,E1 -3510.74,E2 -3510.74} C_VEL
LIN {X 0,Y 544.572,Z 365.459,A -85,B 0,C 180,E1 -3512.219,E2 -3512.219} C_VEL
LIN {X 0,Y 544.651,Z 364.107,A -85,B 0,C 180,E1 -3512.959,E2 -3512.959} C_VEL
LIN {X 0,Y 544.684,Z 361.251,A -85,B 0,C 180,E1 -3514.07,E2 -3514.07} C_VEL
LIN {X 0,Y 544.653,Z 357.382,A -85,B 0,C 180,E1 -3515.183,E2 -3515.183} C_VEL
LIN {X 0,Y 544.769,Z 352.089,A -85,B 0,C 180,E1 -3516.355,E2 -3516.355} C_VEL
LIN {X 0,Y 544.896,Z 344.872,A -85,B 0,C 180,E1 -3517.597,E2 -3517.597} C_VEL
LIN {X 0,Y 545.036,Z 336.739,A -85,B 0,C 180,E1 -3518.715,E2 -3518.715} C_VEL
LIN {X 0,Y 545.216,Z 328.412,A -85,B 0,C 180,E1 -3519.647,E2 -3519.647} C_VEL
LIN {X 0,Y 545.423,Z 319.297,A -85,B 0,C 180,E1 -3520.487,E2 -3520.487} C_VEL
LIN {X 0,Y 545.596,Z 308.755,A -85,B 0,C 180,E1 -3521.276,E2 -3521.276} C_VEL
LIN {X 0,Y 545.852,Z 296.804,A -85,B 0,C 180,E1 -3521.983,E2 -3521.983} C_VEL
LIN {X 0,Y 546.024,Z 284.301,A -85,B 0,C 180,E1 -3522.545,E2 -3522.545} C_VEL
LIN {X 0,Y 546.186,Z 271.787,A -85,B 0,C 180,E1 -3522.943,E2 -3522.943} C_VEL
LIN {X 0,Y 546.305,Z 259.071,A -85,B 0,C 180,E1 -3523.2,E2 -3523.2} C_VEL
LIN {X 0,Y 546.468,Z 163.846,A -85,B 0,C 180,E1 -3524.463,E2 -3524.463} C_VEL
LIN {X 0,Y 545.209,Z 156.926,A -85,B 0,C 180,E1 -3524.599,E2 -3524.599} C_VEL
LIN {X 0,Y 545.394,Z 142.647,A -85,B 0,C 180,E1 -3527.24,E2 -3527.24} C_VEL
LIN {X 0,Y 545.464,Z 133.332,A -85,B 0,C 180,E1 -3528.986,E2 -3528.986} C_VEL
LIN {X 0,Y 545.113,Z 130.586,A -85,B 0,C 180,E1 -3529.536,E2 -3529.536} C_VEL
LIN {X 0,Y 545.049,Z 130.595,A -85,B 0,C 180,E1 -3531.958,E2 -3531.958} C_VEL
LIN {X 0,Y 545.028,Z 130.592,A -85,B 0,C 180,E1 -3534.37,E2 -3534.37} C_VEL
LIN {X 0,Y 545.043,Z 130.588,A -85,B 0,C 180,E1 -3537.162,E2 -3537.162} C_VEL
LIN {X 0,Y 545.044,Z 130.589,A -85,B 0,C 180,E1 -3539.34,E2 -3539.34} C_VEL
LIN {X 0,Y 545.056,Z 130.592,A -85,B 0,C 180,E1 -3541.915,E2 -3541.915} C_VEL
LIN {X 0,Y 545.062,Z 130.585,A -85,B 0,C 180,E1 -3544.564,E2 -3544.564} C_VEL
LIN {X 0,Y 545.031,Z 130.593,A -85,B 0,C 180,E1 -3547.304,E2 -3547.304} C_VEL
LIN {X 0,Y 545.064,Z 130.585,A -85,B 0,C 180,E1 -3550.143,E2 -3550.143} C_VEL
LIN {X 0,Y 545.045,Z 130.591,A -85,B 0,C 180,E1 -3553.11,E2 -3553.11} C_VEL
LIN {X 0,Y 545.045,Z 130.587,A -85,B 0,C 180,E1 -3556.226,E2 -3556.226} C_VEL
LIN {X 0,Y 545.07,Z 130.587,A -85,B 0,C 180,E1 -3558.884,E2 -3558.884} C_VEL
LIN {X 0,Y 545.043,Z 130.588,A -85,B 0,C 180,E1 -3561.864,E2 -3561.864} C_VEL
LIN {X 0,Y 545.023,Z 130.591,A -85,B 0,C 180,E1 -3564.53,E2 -3564.53} C_VEL
LIN {X 0,Y 545.059,Z 130.591,A -85,B 0,C 180,E1 -3567.211,E2 -3567.211} C_VEL
LIN {X 0,Y 545.059,Z 130.585,A -85,B 0,C 180,E1 -3569.81,E2 -3569.81} C_VEL
LIN {X 0,Y 545.053,Z 130.595,A -85,B 0,C 180,E1 -3572.834,E2 -3572.834} C_VEL
LIN {X 0,Y 545.017,Z 130.59,A -85,B 0,C 180,E1 -3575.629,E2 -3575.629} C_VEL
LIN {X 0,Y 545.061,Z 130.587,A -85,B 0,C 180,E1 -3578.18,E2 -3578.18} C_VEL
LIN {X 0,Y 545.099,Z 130.586,A -85,B 0,C 180,E1 -3580.414,E2 -3580.414} C_VEL
LIN {X 0,Y 545.013,Z 130.591,A -85,B 0,C 180,E1 -3583.519,E2 -3583.519} C_VEL
LIN {X 0,Y 545.065,Z 130.585,A -85,B 0,C 180,E1 -3585.819,E2 -3585.819} C_VEL
LIN {X 0,Y 545.112,Z 130.581,A -85,B 0,C 180,E1 -3588.849,E2 -3588.849} C_VEL
LIN {X 0,Y 545.064,Z 130.587,A -85,B 0,C 180,E1 -3591.846,E2 -3591.846} C_VEL
LIN {X 0,Y 545.157,Z 130.574,A -85,B 0,C 180,E1 -3594.822,E2 -3594.822} C_VEL
LIN {X 0,Y 545.186,Z 130.573,A -85,B 0,C 180,E1 -3597.784,E2 -3597.784} C_VEL
LIN {X 0,Y 545.186,Z 130.577,A -85,B 0,C 180,E1 -3600,E2 -3600} C_VEL
LIN {X 0,Y 545.136,Z 130.575,A -85,B 0,C 180,E1 -3602.956,E2 -3602.956} C_VEL
LIN {X 0,Y 545.118,Z 130.587,A -85,B 0,C 180,E1 -3605.92,E2 -3605.92} C_VEL
LIN {X 0,Y 545.06,Z 130.585,A -85,B 0,C 180,E1 -3608.901,E2 -3608.901} C_VEL
LIN {X 0,Y 545.057,Z 130.592,A -85,B 0,C 180,E1 -3611.906,E2 -3611.906} C_VEL
LIN {X 0,Y 545.034,Z 130.589,A -85,B 0,C 180,E1 -3614.945,E2 -3614.945} C_VEL
LIN {X 0,Y 545.037,Z 130.59,A -85,B 0,C 180,E1 -3618.027,E2 -3618.027} C_VEL
LIN {X 0,Y 545.024,Z 130.589,A -85,B 0,C 180,E1 -3620.375,E2 -3620.375} C_VEL
LIN {X 0,Y 544.983,Z 130.595,A -85,B 0,C 180,E1 -3622.76,E2 -3622.76} C_VEL
LIN {X 0,Y 545.028,Z 130.596,A -85,B 0,C 180,E1 -3625.495,E2 -3625.495} C_VEL
LIN {X 0,Y 545.028,Z 130.589,A -85,B 0,C 180,E1 -3628.497,E2 -3628.497} C_VEL
LIN {X 0,Y 545.041,Z 130.59,A -85,B 0,C 180,E1 -3631.676,E2 -3631.676} C_VEL
LIN {X 0,Y 545.042,Z 130.589,A -85,B 0,C 180,E1 -3634.566,E2 -3634.566} C_VEL
LIN {X 0,Y 545.027,Z 130.594,A -85,B 0,C 180,E1 -3637.305,E2 -3637.305} C_VEL
LIN {X 0,Y 545.06,Z 130.585,A -85,B 0,C 180,E1 -3640.143,E2 -3640.143} C_VEL
LIN {X 0,Y 545.016,Z 130.595,A -85,B 0,C 180,E1 -3643.113,E2 -3643.113} C_VEL
LIN {X 0,Y 545.027,Z 130.591,A -85,B 0,C 180,E1 -3646.229,E2 -3646.229} C_VEL
LIN {X 0,Y 545.026,Z 130.595,A -85,B 0,C 180,E1 -3648.881,E2 -3648.881} C_VEL
LIN {X 0,Y 545.074,Z 130.589,A -85,B 0,C 180,E1 -3650.818,E2 -3650.818} C_VEL
LIN {X 0,Y 545.032,Z 130.588,A -85,B 0,C 180,E1 -3653.619,E2 -3653.619} C_VEL
LIN {X 0,Y 545.046,Z 130.594,A -85,B 0,C 180,E1 -3656.327,E2 -3656.327} C_VEL
LIN {X 0,Y 545.063,Z 130.587,A -85,B 0,C 180,E1 -3658.952,E2 -3658.952} C_VEL
LIN {X 0,Y 545.044,Z 130.588,A -85,B 0,C 180,E1 -3661.504,E2 -3661.504} C_VEL
LIN {X 0,Y 545.046,Z 130.594,A -85,B 0,C 180,E1 -3663.998,E2 -3663.998} C_VEL
LIN {X 0,Y 545.07,Z 130.66,A -85,B 0,C 180,E1 -3665.972,E2 -3665.972} C_VEL
LIN {X 0,Y 546.16,Z 137.7,A -85,B 0,C 180,E1 -3667.092,E2 -3667.092} C_VEL
LIN {X 0,Y 545.923,Z 154.784,A -85,B 0,C 180,E1 -3669.66,E2 -3669.66} C_VEL
LIN {X 0,Y 545.566,Z 174.207,A -85,B 0,C 180,E1 -3672.534,E2 -3672.534} C_VEL
LIN {X 0,Y 545.282,Z 192.195,A -85,B 0,C 180,E1 -3675.163,E2 -3675.163} C_VEL
LIN {X 0,Y 545.329,Z 194.085,A -85,B 0,C 180,E1 -3675.44,E2 -3675.44} C_VEL
LIN {X 0,Y 546.476,Z 203.538,A -85,B 0,C 180,E1 -3675.596,E2 -3675.596} C_VEL
LIN {X 0,Y 546.207,Z 302.417,A -85,B 0,C 180,E1 -3676.916,E2 -3676.916} C_VEL
LIN {X 0,Y 546.041,Z 315.712,A -85,B 0,C 180,E1 -3677.243,E2 -3677.243} C_VEL
LIN {X 0,Y 545.874,Z 329.019,A -85,B 0,C 180,E1 -3677.735,E2 -3677.735} C_VEL
LIN {X 0,Y 545.663,Z 341.507,A -85,B 0,C 180,E1 -3678.374,E2 -3678.374} C_VEL
LIN {X 0,Y 545.418,Z 353.099,A -85,B 0,C 180,E1 -3679.137,E2 -3679.137} C_VEL
LIN {X 0,Y 545.234,Z 363.31,A -85,B 0,C 180,E1 -3679.979,E2 -3679.979} C_VEL
LIN {X 0,Y 545.057,Z 372.499,A -85,B 0,C 180,E1 -3680.912,E2 -3680.912} C_VEL
LIN {X 0,Y 544.892,Z 381.454,A -85,B 0,C 180,E1 -3682.03,E2 -3682.03} C_VEL
LIN {X 0,Y 544.752,Z 388.661,A -85,B 0,C 180,E1 -3683.146,E2 -3683.146} C_VEL
LIN {X 0,Y 544.741,Z 395.228,A -85,B 0,C 180,E1 -3684.447,E2 -3684.447} C_VEL
LIN {X 0,Y 544.658,Z 399.57,A -85,B 0,C 180,E1 -3685.559,E2 -3685.559} C_VEL
LIN {X 0,Y 544.669,Z 401.87,A -85,B 0,C 180,E1 -3686.301,E2 -3686.301} C_VEL
LIN {X 0,Y 544.65,Z 403.734,A -85,B 0,C 180,E1 -3687.041,E2 -3687.041} C_VEL
LIN {X 0,Y 544.546,Z 406.125,A -85,B 0,C 180,E1 -3688.521,E2 -3688.521} C_VEL
LIN {X 0,Y 544.542,Z 406.734,A -85,B 0,C 180,E1 -3689.26,E2 -3689.26} C_VEL
LIN {X 0,Y 544.541,Z 406.951,A -85,B 0,C 180,E1 -3690,E2 -3690} C_VEL
LIN {X 0,Y 544.542,Z 406.735,A -85,B 0,C 180,E1 -3690.739,E2 -3690.739} C_VEL
LIN {X 0,Y 544.572,Z 405.133,A -85,B 0,C 180,E1 -3692.218,E2 -3692.218} C_VEL
LIN {X 0,Y 544.65,Z 403.739,A -85,B 0,C 180,E1 -3692.958,E2 -3692.958} C_VEL
LIN {X 0,Y 544.684,Z 400.802,A -85,B 0,C 180,E1 -3694.069,E2 -3694.069} C_VEL
LIN {X 0,Y 544.653,Z 396.823,A -85,B 0,C 180,E1 -3695.182,E2 -3695.182} C_VEL
LIN {X 0,Y 544.729,Z 391.436,A -85,B 0,C 180,E1 -3696.348,E2 -3696.348} C_VEL
LIN {X 0,Y 544.859,Z 384.023,A -85,B 0,C 180,E1 -3697.597,E2 -3697.597} C_VEL
LIN {X 0,Y 545,Z 375.73,A -85,B 0,C 180,E1 -3698.715,E2 -3698.715} C_VEL
LIN {X 0,Y 545.147,Z 367.232,A -85,B 0,C 180,E1 -3699.647,E2 -3699.647} C_VEL
LIN {X 0,Y 545.367,Z 356.733,A -85,B 0,C 180,E1 -3700.581,E2 -3700.581} C_VEL
LIN {X 0,Y 545.576,Z 345.168,A -85,B 0,C 180,E1 -3701.406,E2 -3701.406} C_VEL
LIN {X 0,Y 545.774,Z 334.967,A -85,B 0,C 180,E1 -3701.984,E2 -3701.984} C_VEL
LIN {X 0,Y 545.967,Z 323.299,A -85,B 0,C 180,E1 -3702.498,E2 -3702.498} C_VEL
LIN {X 0,Y 546.11,Z 309.857,A -85,B 0,C 180,E1 -3702.92,E2 -3702.92} C_VEL
LIN {X 0,Y 546.264,Z 296.6,A -85,B 0,C 180,E1 -3703.176,E2 -3703.176} C_VEL
LIN {X 0,Y 546.338,Z 201.081,A -85,B 0,C 180,E1 -3704.44,E2 -3704.44} C_VEL
LIN {X 0,Y 545.321,Z 193.951,A -85,B 0,C 180,E1 -3704.579,E2 -3704.579} C_VEL
LIN {X 0,Y 545.554,Z 174.236,A -85,B 0,C 180,E1 -3707.462,E2 -3707.462} C_VEL
LIN {X 0,Y 545.919,Z 154.79,A -85,B 0,C 180,E1 -3710.339,E2 -3710.339} C_VEL
LIN {X 0,Y 546.158,Z 137.706,A -85,B 0,C 180,E1 -3712.908,E2 -3712.908} C_VEL
LIN {X 0,Y 545.081,Z 130.591,A -85,B 0,C 180,E1 -3714.07,E2 -3714.07} C_VEL
LIN {X 0,Y 545.037,Z 130.592,A -85,B 0,C 180,E1 -3717.161,E2 -3717.161} C_VEL
LIN {X 0,Y 545.059,Z 130.588,A -85,B 0,C 180,E1 -3720.189,E2 -3720.189} C_VEL
LIN {X 0,Y 545.067,Z 130.586,A -85,B 0,C 180,E1 -3723.06,E2 -3723.06} C_VEL
LIN {X 0,Y 545.017,Z 130.596,A -85,B 0,C 180,E1 -3725.67,E2 -3725.67} C_VEL
LIN {X 0,Y 545.042,Z 130.587,A -85,B 0,C 180,E1 -3728.237,E2 -3728.237} C_VEL
LIN {X 0,Y 545.073,Z 130.583,A -85,B 0,C 180,E1 -3730.471,E2 -3730.471} C_VEL
LIN {X 0,Y 545.04,Z 130.594,A -85,B 0,C 180,E1 -3733.109,E2 -3733.109} C_VEL
LIN {X 0,Y 545.039,Z 130.587,A -85,B 0,C 180,E1 -3736.226,E2 -3736.226} C_VEL
LIN {X 0,Y 545.021,Z 130.595,A -85,B 0,C 180,E1 -3738.88,E2 -3738.88} C_VEL
LIN {X 0,Y 545.039,Z 130.588,A -85,B 0,C 180,E1 -3741.761,E2 -3741.761} C_VEL
LIN {X 0,Y 545.016,Z 130.593,A -85,B 0,C 180,E1 -3744.53,E2 -3744.53} C_VEL
LIN {X 0,Y 545.052,Z 130.59,A -85,B 0,C 180,E1 -3747.21,E2 -3747.21} C_VEL
LIN {X 0,Y 545.053,Z 130.586,A -85,B 0,C 180,E1 -3749.81,E2 -3749.81} C_VEL
LIN {X 0,Y 545.026,Z 130.597,A -85,B 0,C 180,E1 -3752.838,E2 -3752.838} C_VEL
LIN {X 0,Y 545.009,Z 130.591,A -85,B 0,C 180,E1 -3755.629,E2 -3755.629} C_VEL
LIN {X 0,Y 545.053,Z 130.589,A -85,B 0,C 180,E1 -3758.18,E2 -3758.18} C_VEL
LIN {X 0,Y 545.091,Z 130.589,A -85,B 0,C 180,E1 -3760.414,E2 -3760.414} C_VEL
LIN {X 0,Y 545.004,Z 130.592,A -85,B 0,C 180,E1 -3763.519,E2 -3763.519} C_VEL
LIN {X 0,Y 545.057,Z 130.587,A -85,B 0,C 180,E1 -3765.819,E2 -3765.819} C_VEL
LIN {X 0,Y 545.061,Z 130.586,A -85,B 0,C 180,E1 -3768.848,E2 -3768.848} C_VEL
LIN {X 0,Y 545.054,Z 130.59,A -85,B 0,C 180,E1 -3771.846,E2 -3771.846} C_VEL
LIN {X 0,Y 545.15,Z 130.574,A -85,B 0,C 180,E1 -3774.822,E2 -3774.822} C_VEL
LIN {X 0,Y 545.181,Z 130.575,A -85,B 0,C 180,E1 -3777.784,E2 -3777.784} C_VEL
LIN {X 0,Y 545.18,Z 130.579,A -85,B 0,C 180,E1 -3780,E2 -3780} C_VEL
LIN {X 0,Y 545.133,Z 130.576,A -85,B 0,C 180,E1 -3782.956,E2 -3782.956} C_VEL
LIN {X 0,Y 545.124,Z 130.584,A -85,B 0,C 180,E1 -3785.92,E2 -3785.92} C_VEL
LIN {X 0,Y 545.082,Z 130.582,A -85,B 0,C 180,E1 -3788.901,E2 -3788.901} C_VEL
LIN {X 0,Y 545.083,Z 130.587,A -85,B 0,C 180,E1 -3791.905,E2 -3791.905} C_VEL
LIN {X 0,Y 545.065,Z 130.586,A -85,B 0,C 180,E1 -3794.944,E2 -3794.944} C_VEL
LIN {X 0,Y 545.036,Z 130.59,A -85,B 0,C 180,E1 -3798.027,E2 -3798.027} C_VEL
LIN {X 0,Y 545.079,Z 130.582,A -85,B 0,C 180,E1 -3800.373,E2 -3800.373} C_VEL
LIN {X 0,Y 545.06,Z 130.59,A -85,B 0,C 180,E1 -3803.56,E2 -3803.56} C_VEL
LIN {X 0,Y 545.047,Z 130.59,A -85,B 0,C 180,E1 -3806.827,E2 -3806.827} C_VEL
LIN {X 0,Y 545.017,Z 130.596,A -85,B 0,C 180,E1 -3809.341,E2 -3809.341} C_VEL
LIN {X 0,Y 545.044,Z 130.587,A -85,B 0,C 180,E1 -3811.916,E2 -3811.916} C_VEL
LIN {X 0,Y 545.05,Z 130.589,A -85,B 0,C 180,E1 -3814.566,E2 -3814.566} C_VEL
LIN {X 0,Y 545.057,Z 130.594,A -85,B 0,C 180,E1 -3816.967,E2 -3816.967} C_VEL
LIN {X 0,Y 544.347,Z 130.677,A -85,B 0,C 180,E1 -3817.584,E2 -3817.584} C_VEL
LIN {X 0,Y 541.481,Z 131.035,A -85,B 0,C 180,E1 -3818.585,E2 -3818.585} C_VEL
LIN {X 0,Y 539.087,Z 131.331,A -85,B 0,C 180,E1 -3819.39,E2 -3819.39} C_VEL
LIN {X 0,Y 538.064,Z 131.457,A -85,B 0,C 180,E1 -3820.012,E2 -3820.012} C_VEL
LIN {X 0,Y 537.982,Z 131.468,A -85,B 0,C 180,E1 -3820.223,E2 -3820.223} C_VEL
LIN {X 0,Y 537.973,Z 131.473,A -85,B 0,C 180,E1 -3822.983,E2 -3822.983} C_VEL
LIN {X 0,Y 538.013,Z 131.463,A -85,B 0,C 180,E1 -3825.928,E2 -3825.928} C_VEL
LIN {X 0,Y 538.018,Z 131.463,A -85,B 0,C 180,E1 -3829.257,E2 -3829.257} C_VEL
LIN {X 0,Y 537.984,Z 131.47,A -85,B 0,C 180,E1 -3832.123,E2 -3832.123} C_VEL
LIN {X 0,Y 537.991,Z 131.468,A -85,B 0,C 180,E1 -3834.916,E2 -3834.916} C_VEL
LIN {X 0,Y 538.015,Z 131.463,A -85,B 0,C 180,E1 -3837.618,E2 -3837.618} C_VEL
LIN {X 0,Y 537.998,Z 131.473,A -85,B 0,C 180,E1 -3840.239,E2 -3840.239} C_VEL
LIN {X 0,Y 538.013,Z 131.464,A -85,B 0,C 180,E1 -3842.794,E2 -3842.794} C_VEL
LIN {X 0,Y 537.986,Z 131.466,A -85,B 0,C 180,E1 -3845.29,E2 -3845.29} C_VEL
LIN {X 0,Y 538.015,Z 131.471,A -85,B 0,C 180,E1 -3848.043,E2 -3848.043} C_VEL
LIN {X 0,Y 538.122,Z 131.612,A -85,B 0,C 180,E1 -3850.498,E2 -3850.498} C_VEL
LIN {X 0,Y 538.505,Z 137.048,A -85,B 0,C 180,E1 -3851.55,E2 -3851.55} C_VEL
LIN {X 0,Y 538.255,Z 153.698,A -85,B 0,C 180,E1 -3854.669,E2 -3854.669} C_VEL
LIN {X 0,Y 538.217,Z 157.107,A -85,B 0,C 180,E1 -3855.299,E2 -3855.299} C_VEL
LIN {X 0,Y 539.721,Z 166.012,A -85,B 0,C 180,E1 -3855.469,E2 -3855.469} C_VEL
LIN {X 0,Y 539.328,Z 263.999,A -85,B 0,C 180,E1 -3856.795,E2 -3856.795} C_VEL
LIN {X 0,Y 539.18,Z 277.185,A -85,B 0,C 180,E1 -3857.126,E2 -3857.126} C_VEL
LIN {X 0,Y 539.003,Z 289.282,A -85,B 0,C 180,E1 -3857.577,E2 -3857.577} C_VEL
LIN {X 0,Y 538.802,Z 300.764,A -85,B 0,C 180,E1 -3858.15,E2 -3858.15} C_VEL
LIN {X 0,Y 538.596,Z 312.357,A -85,B 0,C 180,E1 -3858.904,E2 -3858.904} C_VEL
LIN {X 0,Y 538.345,Z 322.825,A -85,B 0,C 180,E1 -3859.755,E2 -3859.755} C_VEL
LIN {X 0,Y 538.169,Z 331.376,A -85,B 0,C 180,E1 -3860.606,E2 -3860.606} C_VEL
LIN {X 0,Y 537.954,Z 339.251,A -85,B 0,C 180,E1 -3861.549,E2 -3861.549} C_VEL
LIN {X 0,Y 537.812,Z 346.95,A -85,B 0,C 180,E1 -3862.681,E2 -3862.681} C_VEL
LIN {X 0,Y 537.739,Z 354.006,A -85,B 0,C 180,E1 -3863.999,E2 -3863.999} C_VEL
LIN {X 0,Y 537.569,Z 358.715,A -85,B 0,C 180,E1 -3865.126,E2 -3865.126} C_VEL
LIN {X 0,Y 537.591,Z 362.316,A -85,B 0,C 180,E1 -3866.253,E2 -3866.253} C_VEL
LIN {X 0,Y 537.58,Z 364.178,A -85,B 0,C 180,E1 -3867.003,E2 -3867.003} C_VEL
LIN {X 0,Y 537.49,Z 365.587,A -85,B 0,C 180,E1 -3867.752,E2 -3867.752} C_VEL
LIN {X 0,Y 537.45,Z 367.204,A -85,B 0,C 180,E1 -3869.251,E2 -3869.251} C_VEL
LIN {X 0,Y 537.45,Z 367.441,A -85,B 0,C 180,E1 -3870,E2 -3870} C_VEL
LIN {X 0,Y 537.45,Z 367.26,A -85,B 0,C 180,E1 -3870.75,E2 -3870.75} C_VEL
LIN {X 0,Y 537.49,Z 365.717,A -85,B 0,C 180,E1 -3872.248,E2 -3872.248} C_VEL
LIN {X 0,Y 537.58,Z 364.364,A -85,B 0,C 180,E1 -3872.998,E2 -3872.998} C_VEL
LIN {X 0,Y 537.609,Z 361.509,A -85,B 0,C 180,E1 -3874.123,E2 -3874.123} C_VEL
LIN {X 0,Y 537.587,Z 357.638,A -85,B 0,C 180,E1 -3875.251,E2 -3875.251} C_VEL
LIN {X 0,Y 537.704,Z 352.721,A -85,B 0,C 180,E1 -3876.362,E2 -3876.362} C_VEL
LIN {X 0,Y 537.817,Z 346.349,A -85,B 0,C 180,E1 -3877.509,E2 -3877.509} C_VEL
LIN {X 0,Y 537.98,Z 338.47,A -85,B 0,C 180,E1 -3878.641,E2 -3878.641} C_VEL
LIN {X 0,Y 538.213,Z 328.666,A -85,B 0,C 180,E1 -3879.774,E2 -3879.774} C_VEL
LIN {X 0,Y 538.47,Z 318.384,A -85,B 0,C 180,E1 -3880.719,E2 -3880.719} C_VEL
LIN {X 0,Y 538.68,Z 307.153,A -85,B 0,C 180,E1 -3881.547,E2 -3881.547} C_VEL
LIN {X 0,Y 538.926,Z 295.244,A -85,B 0,C 180,E1 -3882.235,E2 -3882.235} C_VEL
LIN {X 0,Y 539.108,Z 283.246,A -85,B 0,C 180,E1 -3882.756,E2 -3882.756} C_VEL
LIN {X 0,Y 539.306,Z 270.194,A -85,B 0,C 180,E1 -3883.159,E2 -3883.159} C_VEL
LIN {X 0,Y 539.428,Z 257.752,A -85,B 0,C 180,E1 -3883.395,E2 -3883.395} C_VEL
LIN {X 0,Y 539.577,Z 164.552,A -85,B 0,C 180,E1 -3884.645,E2 -3884.645} C_VEL
LIN {X 0,Y 538.177,Z 157.117,A -85,B 0,C 180,E1 -3884.792,E2 -3884.792} C_VEL
LIN {X 0,Y 538.391,Z 142.708,A -85,B 0,C 180,E1 -3887.472,E2 -3887.472} C_VEL
LIN {X 0,Y 538.465,Z 134.408,A -85,B 0,C 180,E1 -3889.044,E2 -3889.044} C_VEL
LIN {X 0,Y 538.081,Z 131.463,A -85,B 0,C 180,E1 -3889.653,E2 -3889.653} C_VEL
LIN {X 0,Y 537.994,Z 131.471,A -85,B 0,C 180,E1 -3892.262,E2 -3892.262} C_VEL
LIN {X 0,Y 537.989,Z 131.467,A -85,B 0,C 180,E1 -3894.71,E2 -3894.71} C_VEL
LIN {X 0,Y 538.015,Z 131.464,A -85,B 0,C 180,E1 -3897.343,E2 -3897.343} C_VEL
LIN {X 0,Y 538.008,Z 131.472,A -85,B 0,C 180,E1 -3899.762,E2 -3899.762} C_VEL
LIN {X 0,Y 538.019,Z 131.463,A -85,B 0,C 180,E1 -3902.383,E2 -3902.383} C_VEL
LIN {X 0,Y 537.995,Z 131.467,A -85,B 0,C 180,E1 -3905.084,E2 -3905.084} C_VEL
LIN {X 0,Y 537.988,Z 131.47,A -85,B 0,C 180,E1 -3907.878,E2 -3907.878} C_VEL
LIN {X 0,Y 538.022,Z 131.462,A -85,B 0,C 180,E1 -3910.778,E2 -3910.778} C_VEL
LIN {X 0,Y 538.018,Z 131.463,A -85,B 0,C 180,E1 -3914.073,E2 -3914.073} C_VEL
LIN {X 0,Y 537.979,Z 131.472,A -85,B 0,C 180,E1 -3917.018,E2 -3917.018} C_VEL
LIN {X 0,Y 538.021,Z 131.471,A -85,B 0,C 180,E1 -3919.256,E2 -3919.256} C_VEL
LIN {X 0,Y 537.985,Z 131.466,A -85,B 0,C 180,E1 -3922.121,E2 -3922.121} C_VEL
LIN {X 0,Y 537.985,Z 131.473,A -85,B 0,C 180,E1 -3924.914,E2 -3924.914} C_VEL
LIN {X 0,Y 538.009,Z 131.465,A -85,B 0,C 180,E1 -3927.616,E2 -3927.616} C_VEL
LIN {X 0,Y 537.995,Z 131.466,A -85,B 0,C 180,E1 -3930.237,E2 -3930.237} C_VEL
LIN {X 0,Y 538.023,Z 131.47,A -85,B 0,C 180,E1 -3932.794,E2 -3932.794} C_VEL
LIN {X 0,Y 537.987,Z 131.468,A -85,B 0,C 180,E1 -3935.289,E2 -3935.289} C_VEL
LIN {X 0,Y 538.011,Z 131.464,A -85,B 0,C 180,E1 -3938.042,E2 -3938.042} C_VEL
LIN {X 0,Y 538.003,Z 131.468,A -85,B 0,C 180,E1 -3940.939,E2 -3940.939} C_VEL
LIN {X 0,Y 537.96,Z 131.47,A -85,B 0,C 180,E1 -3943.297,E2 -3943.297} C_VEL
LIN {X 0,Y 538.037,Z 131.46,A -85,B 0,C 180,E1 -3945.63,E2 -3945.63} C_VEL
LIN {X 0,Y 538.072,Z 131.46,A -85,B 0,C 180,E1 -3948.701,E2 -3948.701} C_VEL
LIN {X 0,Y 538.035,Z 131.462,A -85,B 0,C 180,E1 -3951.739,E2 -3951.739} C_VEL
LIN {X 0,Y 538.117,Z 131.452,A -85,B 0,C 180,E1 -3954.754,E2 -3954.754} C_VEL
LIN {X 0,Y 538.157,Z 131.448,A -85,B 0,C 180,E1 -3957.755,E2 -3957.755} C_VEL
LIN {X 0,Y 538.154,Z 131.453,A -85,B 0,C 180,E1 -3960,E2 -3960} C_VEL
LIN {X 0,Y 538.104,Z 131.451,A -85,B 0,C 180,E1 -3962.995,E2 -3962.995} C_VEL
LIN {X 0,Y 538.074,Z 131.463,A -85,B 0,C 180,E1 -3965.998,E2 -3965.998} C_VEL
LIN {X 0,Y 538.019,Z 131.462,A -85,B 0,C 180,E1 -3969.018,E2 -3969.018} C_VEL
LIN {X 0,Y 538.008,Z 131.467,A -85,B 0,C 180,E1 -3972.064,E2 -3972.064} C_VEL
LIN {X 0,Y 537.983,Z 131.469,A -85,B 0,C 180,E1 -3975.146,E2 -3975.146} C_VEL
LIN {X 0,Y 537.99,Z 131.466,A -85,B 0,C 180,E1 -3978.272,E2 -3978.272} C_VEL
LIN {X 0,Y 537.982,Z 131.467,A -85,B 0,C 180,E1 -3980.654,E2 -3980.654} C_VEL
LIN {X 0,Y 537.971,Z 131.472,A -85,B 0,C 180,E1 -3983.074,E2 -3983.074} C_VEL
LIN {X 0,Y 537.987,Z 131.47,A -85,B 0,C 180,E1 -3985.661,E2 -3985.661} C_VEL
LIN {X 0,Y 537.968,Z 131.469,A -85,B 0,C 180,E1 -3988.054,E2 -3988.054} C_VEL
LIN {X 0,Y 537.984,Z 131.468,A -85,B 0,C 180,E1 -3990.629,E2 -3990.629} C_VEL
LIN {X 0,Y 538.017,Z 131.469,A -85,B 0,C 180,E1 -3993.279,E2 -3993.279} C_VEL
LIN {X 0,Y 537.967,Z 131.468,A -85,B 0,C 180,E1 -3996.007,E2 -3996.007} C_VEL
LIN {X 0,Y 538.006,Z 131.471,A -85,B 0,C 180,E1 -3998.831,E2 -3998.831} C_VEL
LIN {X 0,Y 537.986,Z 131.466,A -85,B 0,C 180,E1 -4001.874,E2 -4001.874} C_VEL
LIN {X 0,Y 537.992,Z 131.474,A -85,B 0,C 180,E1 -4004.864,E2 -4004.864} C_VEL
LIN {X 0,Y 537.972,Z 131.47,A -85,B 0,C 180,E1 -4007.21,E2 -4007.21} C_VEL
LIN {X 0,Y 538.028,Z 131.467,A -85,B 0,C 180,E1 -4010.416,E2 -4010.416} C_VEL
LIN {X 0,Y 538.017,Z 131.464,A -85,B 0,C 180,E1 -4013.067,E2 -4013.067} C_VEL
LIN {X 0,Y 537.998,Z 131.466,A -85,B 0,C 180,E1 -4015.825,E2 -4015.825} C_VEL
LIN {X 0,Y 538.009,Z 131.472,A -85,B 0,C 180,E1 -4018.499,E2 -4018.499} C_VEL
LIN {X 0,Y 538.02,Z 131.464,A -85,B 0,C 180,E1 -4021.098,E2 -4021.098} C_VEL
LIN {X 0,Y 537.992,Z 131.469,A -85,B 0,C 180,E1 -4023.631,E2 -4023.631} C_VEL
LIN {X 0,Y 538.034,Z 131.566,A -85,B 0,C 180,E1 -4025.816,E2 -4025.816} C_VEL
LIN {X 0,Y 539.221,Z 138.778,A -85,B 0,C 180,E1 -4026.983,E2 -4026.983} C_VEL
LIN {X 0,Y 538.951,Z 155.571,A -85,B 0,C 180,E1 -4029.542,E2 -4029.542} C_VEL
LIN {X 0,Y 538.559,Z 175.523,A -85,B 0,C 180,E1 -4032.534,E2 -4032.534} C_VEL
LIN {X 0,Y 538.256,Z 192.608,A -85,B 0,C 180,E1 -4035.065,E2 -4035.065} C_VEL
LIN {X 0,Y 538.252,Z 193.823,A -85,B 0,C 180,E1 -4035.244,E2 -4035.244} C_VEL
LIN {X 0,Y 539.593,Z 203.968,A -85,B 0,C 180,E1 -4035.418,E2 -4035.418} C_VEL
LIN {X 0,Y 539.313,Z 302.159,A -85,B 0,C 180,E1 -4036.746,E2 -4036.746} C_VEL
LIN {X 0,Y 539.123,Z 315.453,A -85,B 0,C 180,E1 -4037.076,E2 -4037.076} C_VEL
LIN {X 0,Y 538.889,Z 328.757,A -85,B 0,C 180,E1 -4037.573,E2 -4037.573} C_VEL
LIN {X 0,Y 538.642,Z 341.245,A -85,B 0,C 180,E1 -4038.22,E2 -4038.22} C_VEL
LIN {X 0,Y 538.426,Z 352.839,A -85,B 0,C 180,E1 -4038.995,E2 -4038.995} C_VEL
LIN {X 0,Y 538.213,Z 363.05,A -85,B 0,C 180,E1 -4039.846,E2 -4039.846} C_VEL
LIN {X 0,Y 538.001,Z 372.238,A -85,B 0,C 180,E1 -4040.791,E2 -4040.791} C_VEL
LIN {X 0,Y 537.815,Z 381.193,A -85,B 0,C 180,E1 -4041.924,E2 -4041.924} C_VEL
LIN {X 0,Y 537.679,Z 388.401,A -85,B 0,C 180,E1 -4043.055,E2 -4043.055} C_VEL
LIN {X 0,Y 537.657,Z 394.968,A -85,B 0,C 180,E1 -4044.374,E2 -4044.374} C_VEL
LIN {X 0,Y 537.552,Z 399.31,A -85,B 0,C 180,E1 -4045.501,E2 -4045.501} C_VEL
LIN {X 0,Y 537.591,Z 401.611,A -85,B 0,C 180,E1 -4046.252,E2 -4046.252} C_VEL
LIN {X 0,Y 537.551,Z 403.474,A -85,B 0,C 180,E1 -4047.002,E2 -4047.002} C_VEL
LIN {X 0,Y 537.451,Z 405.866,A -85,B 0,C 180,E1 -4048.501,E2 -4048.501} C_VEL
LIN {X 0,Y 537.446,Z 406.475,A -85,B 0,C 180,E1 -4049.25,E2 -4049.25} C_VEL
LIN {X 0,Y 537.447,Z 406.692,A -85,B 0,C 180,E1 -4050,E2 -4050} C_VEL
LIN {X 0,Y 537.451,Z 405.869,A -85,B 0,C 180,E1 -4051.498,E2 -4051.498} C_VEL
LIN {X 0,Y 537.49,Z 404.874,A -85,B 0,C 180,E1 -4052.248,E2 -4052.248} C_VEL
LIN {X 0,Y 537.551,Z 403.48,A -85,B 0,C 180,E1 -4052.997,E2 -4052.997} C_VEL
LIN {X 0,Y 537.603,Z 400.543,A -85,B 0,C 180,E1 -4054.123,E2 -4054.123} C_VEL
LIN {X 0,Y 537.587,Z 396.563,A -85,B 0,C 180,E1 -4055.25,E2 -4055.25} C_VEL
LIN {X 0,Y 537.653,Z 390.472,A -85,B 0,C 180,E1 -4056.563,E2 -4056.563} C_VEL
LIN {X 0,Y 537.783,Z 383.763,A -85,B 0,C 180,E1 -4057.697,E2 -4057.697} C_VEL
LIN {X 0,Y 537.933,Z 375.469,A -85,B 0,C 180,E1 -4058.83,E2 -4058.83} C_VEL
LIN {X 0,Y 538.102,Z 366.971,A -85,B 0,C 180,E1 -4059.775,E2 -4059.775} C_VEL
LIN {X 0,Y 538.362,Z 356.473,A -85,B 0,C 180,E1 -4060.72,E2 -4060.72} C_VEL
LIN {X 0,Y 538.581,Z 345.289,A -85,B 0,C 180,E1 -4061.531,E2 -4061.531} C_VEL
LIN {X 0,Y 538.814,Z 334.707,A -85,B 0,C 180,E1 -4062.141,E2 -4062.141} C_VEL
LIN {X 0,Y 539.016,Z 323.039,A -85,B 0,C 180,E1 -4062.662,E2 -4062.662} C_VEL
LIN {X 0,Y 539.186,Z 310.514,A -85,B 0,C 180,E1 -4063.065,E2 -4063.065} C_VEL
LIN {X 0,Y 539.349,Z 297.854,A -85,B 0,C 180,E1 -4063.325,E2 -4063.325} C_VEL
LIN {X 0,Y 539.505,Z 202.142,A -85,B 0,C 180,E1 -4064.609,E2 -4064.609} C_VEL
LIN {X 0,Y 538.296,Z 193.746,A -85,B 0,C 180,E1 -4064.766,E2 -4064.766} C_VEL
LIN {X 0,Y 538.548,Z 175.527,A -85,B 0,C 180,E1 -4067.466,E2 -4067.466} C_VEL
LIN {X 0,Y 538.964,Z 155.576,A -85,B 0,C 180,E1 -4070.457,E2 -4070.457} C_VEL
LIN {X 0,Y 539.207,Z 138.784,A -85,B 0,C 180,E1 -4073.017,E2 -4073.017} C_VEL
LIN {X 0,Y 538.047,Z 131.466,A -85,B 0,C 180,E1 -4074.21,E2 -4074.21} C_VEL
LIN {X 0,Y 538.008,Z 131.47,A -85,B 0,C 180,E1 -4077.341,E2 -4077.341} C_VEL
LIN {X 0,Y 537.997,Z 131.473,A -85,B 0,C 180,E1 -4079.761,E2 -4079.761} C_VEL
LIN {X 0,Y 538.011,Z 131.463,A -85,B 0,C 180,E1 -4082.382,E2 -4082.382} C_VEL
LIN {X 0,Y 537.983,Z 131.47,A -85,B 0,C 180,E1 -4085.084,E2 -4085.084} C_VEL
LIN {X 0,Y 537.982,Z 131.469,A -85,B 0,C 180,E1 -4087.877,E2 -4087.877} C_VEL
LIN {X 0,Y 538,Z 131.466,A -85,B 0,C 180,E1 -4090.741,E2 -4090.741} C_VEL
LIN {X 0,Y 537.997,Z 131.466,A -85,B 0,C 180,E1 -4093.815,E2 -4093.815} C_VEL
LIN {X 0,Y 537.992,Z 131.465,A -85,B 0,C 180,E1 -4096.183,E2 -4096.183} C_VEL
LIN {X 0,Y 537.998,Z 131.471,A -85,B 0,C 180,E1 -4099.257,E2 -4099.257} C_VEL
LIN {X 0,Y 537.979,Z 131.467,A -85,B 0,C 180,E1 -4102.121,E2 -4102.121} C_VEL
LIN {X 0,Y 537.978,Z 131.476,A -85,B 0,C 180,E1 -4104.914,E2 -4104.914} C_VEL
LIN {X 0,Y 538.002,Z 131.465,A -85,B 0,C 180,E1 -4107.616,E2 -4107.616} C_VEL
LIN {X 0,Y 537.988,Z 131.468,A -85,B 0,C 180,E1 -4110.237,E2 -4110.237} C_VEL
LIN {X 0,Y 537.999,Z 131.473,A -85,B 0,C 180,E1 -4112.793,E2 -4112.793} C_VEL
LIN {X 0,Y 537.972,Z 131.469,A -85,B 0,C 180,E1 -4115.289,E2 -4115.289} C_VEL
LIN {X 0,Y 538,Z 131.466,A -85,B 0,C 180,E1 -4118.043,E2 -4118.043} C_VEL
LIN {X 0,Y 537.994,Z 131.468,A -85,B 0,C 180,E1 -4120.938,E2 -4120.938} C_VEL
LIN {X 0,Y 537.952,Z 131.47,A -85,B 0,C 180,E1 -4123.297,E2 -4123.297} C_VEL
LIN {X 0,Y 538.029,Z 131.461,A -85,B 0,C 180,E1 -4125.63,E2 -4125.63} C_VEL
LIN {X 0,Y 538.013,Z 131.466,A -85,B 0,C 180,E1 -4128.7,E2 -4128.7} C_VEL
LIN {X 0,Y 538.022,Z 131.464,A -85,B 0,C 180,E1 -4131.739,E2 -4131.739} C_VEL
LIN {X 0,Y 538.11,Z 131.452,A -85,B 0,C 180,E1 -4134.754,E2 -4134.754} C_VEL
LIN {X 0,Y 538.152,Z 131.45,A -85,B 0,C 180,E1 -4137.755,E2 -4137.755} C_VEL
LIN {X 0,Y 538.149,Z 131.455,A -85,B 0,C 180,E1 -4140,E2 -4140} C_VEL
LIN {X 0,Y 538.1,Z 131.452,A -85,B 0,C 180,E1 -4142.995,E2 -4142.995} C_VEL
LIN {X 0,Y 538.08,Z 131.46,A -85,B 0,C 180,E1 -4145.998,E2 -4145.998} C_VEL
LIN {X 0,Y 538.035,Z 131.461,A -85,B 0,C 180,E1 -4149.018,E2 -4149.018} C_VEL
LIN {X 0,Y 538.042,Z 131.462,A -85,B 0,C 180,E1 -4152.064,E2 -4152.064} C_VEL
LIN {X 0,Y 538.025,Z 131.464,A -85,B 0,C 180,E1 -4155.144,E2 -4155.144} C_VEL
LIN {X 0,Y 537.992,Z 131.465,A -85,B 0,C 180,E1 -4158.272,E2 -4158.272} C_VEL
LIN {X 0,Y 538.025,Z 131.462,A -85,B 0,C 180,E1 -4160.652,E2 -4160.652} C_VEL
LIN {X 0,Y 537.996,Z 131.466,A -85,B 0,C 180,E1 -4163.878,E2 -4163.878} C_VEL
LIN {X 0,Y 537.981,Z 131.467,A -85,B 0,C 180,E1 -4166.37,E2 -4166.37} C_VEL
LIN {X 0,Y 537.983,Z 131.472,A -85,B 0,C 180,E1 -4168.926,E2 -4168.926} C_VEL
LIN {X 0,Y 537.999,Z 131.465,A -85,B 0,C 180,E1 -4171.887,E2 -4171.887} C_VEL
LIN {X 0,Y 538,Z 131.468,A -85,B 0,C 180,E1 -4174.618,E2 -4174.618} C_VEL
LIN {X 0,Y 537.996,Z 131.47,A -85,B 0,C 180,E1 -4177.17,E2 -4177.17} C_VEL
LIN {X 0,Y 538.001,Z 131.464,A -85,B 0,C 180,E1 -4179.799,E2 -4179.799} C_VEL
LIN {X 0,Y 537.982,Z 131.468,A -85,B 0,C 180,E1 -4180.223,E2 -4180.223} C_VEL
LIN {X 0,Y 537.319,Z 131.558,A -85,B 0,C 180,E1 -4180.848,E2 -4180.848} C_VEL
LIN {X 0,Y 534.47,Z 131.911,A -85,B 0,C 180,E1 -4181.863,E2 -4181.863} C_VEL
LIN {X 0,Y 532.057,Z 132.212,A -85,B 0,C 180,E1 -4182.68,E2 -4182.68} C_VEL
LIN {X 0,Y 531.017,Z 132.336,A -85,B 0,C 180,E1 -4183.311,E2 -4183.311} C_VEL
LIN {X 0,Y 530.93,Z 132.345,A -85,B 0,C 180,E1 -4183.524,E2 -4183.524} C_VEL
LIN {X 0,Y 530.939,Z 132.35,A -85,B 0,C 180,E1 -4186.504,E2 -4186.504} C_VEL
LIN {X 0,Y 530.957,Z 132.345,A -85,B 0,C 180,E1 -4188.98,E2 -4188.98} C_VEL
LIN {X 0,Y 530.949,Z 132.343,A -85,B 0,C 180,E1 -4191.53,E2 -4191.53} C_VEL
LIN {X 0,Y 530.947,Z 132.351,A -85,B 0,C 180,E1 -4194.38,E2 -4194.38} C_VEL
LIN {X 0,Y 530.964,Z 132.341,A -85,B 0,C 180,E1 -4197.134,E2 -4197.134} C_VEL
LIN {X 0,Y 530.949,Z 132.345,A -85,B 0,C 180,E1 -4199.803,E2 -4199.803} C_VEL
LIN {X 0,Y 530.964,Z 132.346,A -85,B 0,C 180,E1 -4202.478,E2 -4202.478} C_VEL
LIN {X 0,Y 530.956,Z 132.342,A -85,B 0,C 180,E1 -4204.941,E2 -4204.941} C_VEL
LIN {X 0,Y 530.977,Z 132.346,A -85,B 0,C 180,E1 -4207.899,E2 -4207.899} C_VEL
LIN {X 0,Y 531.055,Z 132.458,A -85,B 0,C 180,E1 -4210.383,E2 -4210.383} C_VEL
LIN {X 0,Y 531.515,Z 137.099,A -85,B 0,C 180,E1 -4211.299,E2 -4211.299} C_VEL
LIN {X 0,Y 531.285,Z 151.729,A -85,B 0,C 180,E1 -4214.069,E2 -4214.069} C_VEL
LIN {X 0,Y 531.238,Z 157.304,A -85,B 0,C 180,E1 -4215.104,E2 -4215.104} C_VEL
LIN {X 0,Y 532.853,Z 166.028,A -85,B 0,C 180,E1 -4215.273,E2 -4215.273} C_VEL
LIN {X 0,Y 532.442,Z 264.286,A -85,B 0,C 180,E1 -4216.621,E2 -4216.621} C_VEL
LIN {X 0,Y 532.279,Z 277.463,A -85,B 0,C 180,E1 -4216.957,E2 -4216.957} C_VEL
LIN {X 0,Y 532.075,Z 289.555,A -85,B 0,C 180,E1 -4217.412,E2 -4217.412} C_VEL
LIN {X 0,Y 531.857,Z 301.279,A -85,B 0,C 180,E1 -4218.008,E2 -4218.008} C_VEL
LIN {X 0,Y 531.645,Z 312.624,A -85,B 0,C 180,E1 -4218.757,E2 -4218.757} C_VEL
LIN {X 0,Y 531.369,Z 323.091,A -85,B 0,C 180,E1 -4219.619,E2 -4219.619} C_VEL
LIN {X 0,Y 531.149,Z 331.641,A -85,B 0,C 180,E1 -4220.48,E2 -4220.48} C_VEL
LIN {X 0,Y 530.944,Z 339.514,A -85,B 0,C 180,E1 -4221.437,E2 -4221.437} C_VEL
LIN {X 0,Y 530.752,Z 347.213,A -85,B 0,C 180,E1 -4222.583,E2 -4222.583} C_VEL
LIN {X 0,Y 530.674,Z 354.268,A -85,B 0,C 180,E1 -4223.919,E2 -4223.919} C_VEL
LIN {X 0,Y 530.486,Z 358.976,A -85,B 0,C 180,E1 -4225.06,E2 -4225.06} C_VEL
LIN {X 0,Y 530.517,Z 362.576,A -85,B 0,C 180,E1 -4226.203,E2 -4226.203} C_VEL
LIN {X 0,Y 530.512,Z 364.438,A -85,B 0,C 180,E1 -4226.963,E2 -4226.963} C_VEL
LIN {X 0,Y 530.412,Z 365.847,A -85,B 0,C 180,E1 -4227.722,E2 -4227.722} C_VEL
LIN {X 0,Y 530.355,Z 367.463,A -85,B 0,C 180,E1 -4229.241,E2 -4229.241} C_VEL
LIN {X 0,Y 530.355,Z 367.701,A -85,B 0,C 180,E1 -4230,E2 -4230} C_VEL
LIN {X 0,Y 530.355,Z 367.519,A -85,B 0,C 180,E1 -4230.76,E2 -4230.76} C_VEL
LIN {X 0,Y 530.413,Z 365.975,A -85,B 0,C 180,E1 -4232.278,E2 -4232.278} C_VEL
LIN {X 0,Y 530.512,Z 364.621,A -85,B 0,C 180,E1 -4233.038,E2 -4233.038} C_VEL
LIN {X 0,Y 530.537,Z 361.766,A -85,B 0,C 180,E1 -4234.179,E2 -4234.179} C_VEL
LIN {X 0,Y 530.524,Z 357.895,A -85,B 0,C 180,E1 -4235.321,E2 -4235.321} C_VEL
LIN {X 0,Y 530.627,Z 352.184,A -85,B 0,C 180,E1 -4236.607,E2 -4236.607} C_VEL
LIN {X 0,Y 530.816,Z 345.384,A -85,B 0,C 180,E1 -4237.8,E2 -4237.8} C_VEL
LIN {X 0,Y 530.996,Z 337.248,A -85,B 0,C 180,E1 -4238.947,E2 -4238.947} C_VEL
LIN {X 0,Y 531.219,Z 328.919,A -85,B 0,C 180,E1 -4239.904,E2 -4239.904} C_VEL
LIN {X 0,Y 531.486,Z 318.636,A -85,B 0,C 180,E1 -4240.862,E2 -4240.862} C_VEL
LIN {X 0,Y 531.733,Z 307.754,A -85,B 0,C 180,E1 -4241.676,E2 -4241.676} C_VEL
LIN {X 0,Y 531.99,Z 297.299,A -85,B 0,C 180,E1 -4242.3,E2 -4242.3} C_VEL
LIN {X 0,Y 532.2,Z 284.785,A -85,B 0,C 180,E1 -4242.876,E2 -4242.876} C_VEL
LIN {X 0,Y 532.389,Z 272.258,A -85,B 0,C 180,E1 -4243.284,E2 -4243.284} C_VEL
LIN {X 0,Y 532.54,Z 259.511,A -85,B 0,C 180,E1 -4243.548,E2 -4243.548} C_VEL
LIN {X 0,Y 532.684,Z 165.221,A -85,B 0,C 180,E1 -4244.833,E2 -4244.833} C_VEL
LIN {X 0,Y 531.184,Z 157.316,A -85,B 0,C 180,E1 -4244.986,E2 -4244.986} C_VEL
LIN {X 0,Y 531.426,Z 142.342,A -85,B 0,C 180,E1 -4247.789,E2 -4247.789} C_VEL
LIN {X 0,Y 531.464,Z 135.486,A -85,B 0,C 180,E1 -4249.104,E2 -4249.104} C_VEL
LIN {X 0,Y 531.061,Z 132.337,A -85,B 0,C 180,E1 -4249.743,E2 -4249.743} C_VEL
LIN {X 0,Y 530.945,Z 132.345,A -85,B 0,C 180,E1 -4252.573,E2 -4252.573} C_VEL
LIN {X 0,Y 530.959,Z 132.342,A -85,B 0,C 180,E1 -4255.06,E2 -4255.06} C_VEL
LIN {X 0,Y 530.967,Z 132.345,A -85,B 0,C 180,E1 -4257.598,E2 -4257.598} C_VEL
LIN {X 0,Y 530.955,Z 132.345,A -85,B 0,C 180,E1 -4260.198,E2 -4260.198} C_VEL
LIN {X 0,Y 530.968,Z 132.34,A -85,B 0,C 180,E1 -4262.866,E2 -4262.866} C_VEL
LIN {X 0,Y 530.951,Z 132.352,A -85,B 0,C 180,E1 -4265.62,E2 -4265.62} C_VEL
LIN {X 0,Y 530.963,Z 132.341,A -85,B 0,C 180,E1 -4268.653,E2 -4268.653} C_VEL
LIN {X 0,Y 530.979,Z 132.348,A -85,B 0,C 180,E1 -4271.437,E2 -4271.437} C_VEL
LIN {X 0,Y 530.971,Z 132.34,A -85,B 0,C 180,E1 -4274.548,E2 -4274.548} C_VEL
LIN {X 0,Y 530.966,Z 132.342,A -85,B 0,C 180,E1 -4277.836,E2 -4277.836} C_VEL
LIN {X 0,Y 530.968,Z 132.341,A -85,B 0,C 180,E1 -4280.555,E2 -4280.555} C_VEL
LIN {X 0,Y 530.948,Z 132.347,A -85,B 0,C 180,E1 -4283.441,E2 -4283.441} C_VEL
LIN {X 0,Y 530.959,Z 132.343,A -85,B 0,C 180,E1 -4286.5,E2 -4286.5} C_VEL
LIN {X 0,Y 530.953,Z 132.345,A -85,B 0,C 180,E1 -4289.358,E2 -4289.358} C_VEL
LIN {X 0,Y 530.966,Z 132.344,A -85,B 0,C 180,E1 -4292.477,E2 -4292.477} C_VEL
LIN {X 0,Y 530.956,Z 132.349,A -85,B 0,C 180,E1 -4294.94,E2 -4294.94} C_VEL
LIN {X 0,Y 530.973,Z 132.34,A -85,B 0,C 180,E1 -4297.898,E2 -4297.898} C_VEL
LIN {X 0,Y 530.966,Z 132.349,A -85,B 0,C 180,E1 -4300.676,E2 -4300.676} C_VEL
LIN {X 0,Y 530.924,Z 132.348,A -85,B 0,C 180,E1 -4303.069,E2 -4303.069} C_VEL
LIN {X 0,Y 530.997,Z 132.337,A -85,B 0,C 180,E1 -4305.435,E2 -4305.435} C_VEL
LIN {X 0,Y 531.03,Z 132.339,A -85,B 0,C 180,E1 -4308.55,E2 -4308.55} C_VEL
LIN {X 0,Y 530.985,Z 132.339,A -85,B 0,C 180,E1 -4311.628,E2 -4311.628} C_VEL
LIN {X 0,Y 531.078,Z 132.329,A -85,B 0,C 180,E1 -4314.685,E2 -4314.685} C_VEL
LIN {X 0,Y 531.129,Z 132.323,A -85,B 0,C 180,E1 -4317.725,E2 -4317.725} C_VEL
LIN {X 0,Y 531.123,Z 132.329,A -85,B 0,C 180,E1 -4320,E2 -4320} C_VEL
LIN {X 0,Y 531.128,Z 132.325,A -85,B 0,C 180,E1 -4322.275,E2 -4322.275} C_VEL
LIN {X 0,Y 531.075,Z 132.328,A -85,B 0,C 180,E1 -4325.315,E2 -4325.315} C_VEL
LIN {X 0,Y 530.976,Z 132.341,A -85,B 0,C 180,E1 -4328.372,E2 -4328.372} C_VEL
LIN {X 0,Y 531.006,Z 132.343,A -85,B 0,C 180,E1 -4331.65,E2 -4331.65} C_VEL
LIN {X 0,Y 530.959,Z 132.342,A -85,B 0,C 180,E1 -4334.928,E2 -4334.928} C_VEL
LIN {X 0,Y 530.966,Z 132.347,A -85,B 0,C 180,E1 -4337.724,E2 -4337.724} C_VEL
LIN {X 0,Y 530.967,Z 132.342,A -85,B 0,C 180,E1 -4340.129,E2 -4340.129} C_VEL
LIN {X 0,Y 530.912,Z 132.347,A -85,B 0,C 180,E1 -4342.575,E2 -4342.575} C_VEL
LIN {X 0,Y 530.94,Z 132.348,A -85,B 0,C 180,E1 -4345.061,E2 -4345.061} C_VEL
LIN {X 0,Y 530.947,Z 132.347,A -85,B 0,C 180,E1 -4347.599,E2 -4347.599} C_VEL
LIN {X 0,Y 530.938,Z 132.346,A -85,B 0,C 180,E1 -4350.639,E2 -4350.639} C_VEL
LIN {X 0,Y 530.958,Z 132.345,A -85,B 0,C 180,E1 -4353.5,E2 -4353.5} C_VEL
LIN {X 0,Y 530.941,Z 132.346,A -85,B 0,C 180,E1 -4356.56,E2 -4356.56} C_VEL
LIN {X 0,Y 530.966,Z 132.343,A -85,B 0,C 180,E1 -4359.445,E2 -4359.445} C_VEL
LIN {X 0,Y 530.917,Z 132.35,A -85,B 0,C 180,E1 -4362.463,E2 -4362.463} C_VEL
LIN {X 0,Y 530.962,Z 132.342,A -85,B 0,C 180,E1 -4365.451,E2 -4365.451} C_VEL
LIN {X 0,Y 530.957,Z 132.349,A -85,B 0,C 180,E1 -4368.561,E2 -4368.561} C_VEL
LIN {X 0,Y 530.949,Z 132.343,A -85,B 0,C 180,E1 -4371.529,E2 -4371.529} C_VEL
LIN {X 0,Y 530.947,Z 132.35,A -85,B 0,C 180,E1 -4374.379,E2 -4374.379} C_VEL
LIN {X 0,Y 530.966,Z 132.341,A -85,B 0,C 180,E1 -4377.133,E2 -4377.133} C_VEL
LIN {X 0,Y 530.951,Z 132.346,A -85,B 0,C 180,E1 -4379.802,E2 -4379.802} C_VEL
LIN {X 0,Y 530.966,Z 132.349,A -85,B 0,C 180,E1 -4382.478,E2 -4382.478} C_VEL
LIN {X 0,Y 530.989,Z 132.401,A -85,B 0,C 180,E1 -4385.646,E2 -4385.646} C_VEL
LIN {X 0,Y 532.265,Z 139.852,A -85,B 0,C 180,E1 -4386.87,E2 -4386.87} C_VEL
LIN {X 0,Y 531.98,Z 156.999,A -85,B 0,C 180,E1 -4389.519,E2 -4389.519} C_VEL
LIN {X 0,Y 531.553,Z 176.581,A -85,B 0,C 180,E1 -4392.495,E2 -4392.495} C_VEL
LIN {X 0,Y 531.209,Z 193.493,A -85,B 0,C 180,E1 -4395.035,E2 -4395.035} C_VEL
LIN {X 0,Y 532.731,Z 204.013,A -85,B 0,C 180,E1 -4395.23,E2 -4395.23} C_VEL
LIN {X 0,Y 532.419,Z 301.9,A -85,B 0,C 180,E1 -4396.571,E2 -4396.571} C_VEL
LIN {X 0,Y 532.209,Z 315.193,A -85,B 0,C 180,E1 -4396.906,E2 -4396.906} C_VEL
LIN {X 0,Y 531.925,Z 328.497,A -85,B 0,C 180,E1 -4397.408,E2 -4397.408} C_VEL
LIN {X 0,Y 531.683,Z 340.849,A -85,B 0,C 180,E1 -4398.056,E2 -4398.056} C_VEL
LIN {X 0,Y 531.449,Z 352.579,A -85,B 0,C 180,E1 -4398.848,E2 -4398.848} C_VEL
LIN {X 0,Y 531.148,Z 362.788,A -85,B 0,C 180,E1 -4399.71,E2 -4399.71} C_VEL
LIN {X 0,Y 530.963,Z 371.978,A -85,B 0,C 180,E1 -4400.668,E2 -4400.668} C_VEL
LIN {X 0,Y 530.764,Z 380.933,A -85,B 0,C 180,E1 -4401.816,E2 -4401.816} C_VEL
LIN {X 0,Y 530.622,Z 388.141,A -85,B 0,C 180,E1 -4402.962,E2 -4402.962} C_VEL
LIN {X 0,Y 530.571,Z 394.708,A -85,B 0,C 180,E1 -4404.298,E2 -4404.298} C_VEL
LIN {X 0,Y 530.45,Z 399.05,A -85,B 0,C 180,E1 -4405.44,E2 -4405.44} C_VEL
LIN {X 0,Y 530.516,Z 401.353,A -85,B 0,C 180,E1 -4406.202,E2 -4406.202} C_VEL
LIN {X 0,Y 530.457,Z 403.215,A -85,B 0,C 180,E1 -4406.962,E2 -4406.962} C_VEL
LIN {X 0,Y 530.411,Z 404.612,A -85,B 0,C 180,E1 -4407.722,E2 -4407.722} C_VEL
LIN {X 0,Y 530.351,Z 406.216,A -85,B 0,C 180,E1 -4409.24,E2 -4409.24} C_VEL
LIN {X 0,Y 530.352,Z 406.433,A -85,B 0,C 180,E1 -4410,E2 -4410} C_VEL
LIN {X 0,Y 530.361,Z 405.61,A -85,B 0,C 180,E1 -4411.518,E2 -4411.518} C_VEL
LIN {X 0,Y 530.411,Z 404.616,A -85,B 0,C 180,E1 -4412.278,E2 -4412.278} C_VEL
LIN {X 0,Y 530.457,Z 403.22,A -85,B 0,C 180,E1 -4413.037,E2 -4413.037} C_VEL
LIN {X 0,Y 530.521,Z 400.284,A -85,B 0,C 180,E1 -4414.178,E2 -4414.178} C_VEL
LIN {X 0,Y 530.521,Z 396.304,A -85,B 0,C 180,E1 -4415.32,E2 -4415.32} C_VEL
LIN {X 0,Y 530.554,Z 390.798,A -85,B 0,C 180,E1 -4416.54,E2 -4416.54} C_VEL
LIN {X 0,Y 530.704,Z 383.502,A -85,B 0,C 180,E1 -4417.801,E2 -4417.801} C_VEL
LIN {X 0,Y 530.886,Z 375.209,A -85,B 0,C 180,E1 -4418.948,E2 -4418.948} C_VEL
LIN {X 0,Y 531.062,Z 366.71,A -85,B 0,C 180,E1 -4419.906,E2 -4419.906} C_VEL
LIN {X 0,Y 531.349,Z 356.212,A -85,B 0,C 180,E1 -4420.864,E2 -4420.864} C_VEL
LIN {X 0,Y 531.609,Z 344.422,A -85,B 0,C 180,E1 -4421.725,E2 -4421.725} C_VEL
LIN {X 0,Y 531.897,Z 332.524,A -85,B 0,C 180,E1 -4422.398,E2 -4422.398} C_VEL
LIN {X 0,Y 532.097,Z 320.173,A -85,B 0,C 180,E1 -4422.927,E2 -4422.927} C_VEL
LIN {X 0,Y 532.296,Z 307.507,A -85,B 0,C 180,E1 -4423.31,E2 -4423.31} C_VEL
LIN {X 0,Y 532.494,Z 294.31,A -85,B 0,C 180,E1 -4423.548,E2 -4423.548} C_VEL
LIN {X 0,Y 532.629,Z 202.722,A -85,B 0,C 180,E1 -4424.791,E2 -4424.791} C_VEL
LIN {X 0,Y 531.273,Z 193.455,A -85,B 0,C 180,E1 -4424.97,E2 -4424.97} C_VEL
LIN {X 0,Y 531.595,Z 174.33,A -85,B 0,C 180,E1 -4427.846,E2 -4427.846} C_VEL
LIN {X 0,Y 532.002,Z 154.305,A -85,B 0,C 180,E1 -4430.896,E2 -4430.896} C_VEL
LIN {X 0,Y 532.252,Z 139.856,A -85,B 0,C 180,E1 -4433.13,E2 -4433.13} C_VEL
LIN {X 0,Y 530.988,Z 132.344,A -85,B 0,C 180,E1 -4434.379,E2 -4434.379} C_VEL
LIN {X 0,Y 530.962,Z 132.348,A -85,B 0,C 180,E1 -4437.521,E2 -4437.521} C_VEL
LIN {X 0,Y 530.958,Z 132.343,A -85,B 0,C 180,E1 -4440.642,E2 -4440.642} C_VEL
LIN {X 0,Y 530.957,Z 132.35,A -85,B 0,C 180,E1 -4443.498,E2 -4443.498} C_VEL
LIN {X 0,Y 530.945,Z 132.343,A -85,B 0,C 180,E1 -4446.558,E2 -4446.558} C_VEL
LIN {X 0,Y 530.978,Z 132.347,A -85,B 0,C 180,E1 -4449.443,E2 -4449.443} C_VEL
LIN {X 0,Y 530.932,Z 132.345,A -85,B 0,C 180,E1 -4452.46,E2 -4452.46} C_VEL
LIN {X 0,Y 530.961,Z 132.346,A -85,B 0,C 180,E1 -4455.45,E2 -4455.45} C_VEL
LIN {X 0,Y 530.952,Z 132.344,A -85,B 0,C 180,E1 -4458.56,E2 -4458.56} C_VEL
LIN {X 0,Y 530.944,Z 132.346,A -85,B 0,C 180,E1 -4461.528,E2 -4461.528} C_VEL
LIN {X 0,Y 530.938,Z 132.346,A -85,B 0,C 180,E1 -4464.379,E2 -4464.379} C_VEL
LIN {X 0,Y 530.956,Z 132.347,A -85,B 0,C 180,E1 -4467.132,E2 -4467.132} C_VEL
LIN {X 0,Y 530.937,Z 132.344,A -85,B 0,C 180,E1 -4469.801,E2 -4469.801} C_VEL
LIN {X 0,Y 530.953,Z 132.347,A -85,B 0,C 180,E1 -4472.478,E2 -4472.478} C_VEL
LIN {X 0,Y 530.939,Z 132.349,A -85,B 0,C 180,E1 -4474.939,E2 -4474.939} C_VEL
LIN {X 0,Y 530.961,Z 132.342,A -85,B 0,C 180,E1 -4477.899,E2 -4477.899} C_VEL
LIN {X 0,Y 530.951,Z 132.349,A -85,B 0,C 180,E1 -4480.676,E2 -4480.676} C_VEL
LIN {X 0,Y 530.916,Z 132.348,A -85,B 0,C 180,E1 -4483.069,E2 -4483.069} C_VEL
LIN {X 0,Y 530.99,Z 132.338,A -85,B 0,C 180,E1 -4485.435,E2 -4485.435} C_VEL
LIN {X 0,Y 530.975,Z 132.344,A -85,B 0,C 180,E1 -4488.548,E2 -4488.548} C_VEL
LIN {X 0,Y 530.971,Z 132.342,A -85,B 0,C 180,E1 -4491.628,E2 -4491.628} C_VEL
LIN {X 0,Y 531.071,Z 132.329,A -85,B 0,C 180,E1 -4494.685,E2 -4494.685} C_VEL
LIN {X 0,Y 531.123,Z 132.325,A -85,B 0,C 180,E1 -4497.725,E2 -4497.725} C_VEL
LIN {X 0,Y 531.117,Z 132.331,A -85,B 0,C 180,E1 -4500,E2 -4500} C_VEL
LIN {X 0,Y 531.124,Z 132.325,A -85,B 0,C 180,E1 -4502.275,E2 -4502.275} C_VEL
LIN {X 0,Y 531.076,Z 132.329,A -85,B 0,C 180,E1 -4505.315,E2 -4505.315} C_VEL
LIN {X 0,Y 531.02,Z 132.335,A -85,B 0,C 180,E1 -4508.371,E2 -4508.371} C_VEL
LIN {X 0,Y 531.038,Z 132.34,A -85,B 0,C 180,E1 -4511.671,E2 -4511.671} C_VEL
LIN {X 0,Y 531.009,Z 132.337,A -85,B 0,C 180,E1 -4514.951,E2 -4514.951} C_VEL
LIN {X 0,Y 530.956,Z 132.342,A -85,B 0,C 180,E1 -4518.523,E2 -4518.523} C_VEL
LIN {X 0,Y 530.987,Z 132.341,A -85,B 0,C 180,E1 -4520.939,E2 -4520.939} C_VEL
LIN {X 0,Y 530.94,Z 132.344,A -85,B 0,C 180,E1 -4524.227,E2 -4524.227} C_VEL
LIN {X 0,Y 530.947,Z 132.345,A -85,B 0,C 180,E1 -4526.747,E2 -4526.747} C_VEL
LIN {X 0,Y 530.952,Z 132.349,A -85,B 0,C 180,E1 -4529.325,E2 -4529.325} C_VEL
LIN {X 0,Y 530.954,Z 132.342,A -85,B 0,C 180,E1 -4532.1,E2 -4532.1} C_VEL
LIN {X 0,Y 530.959,Z 132.348,A -85,B 0,C 180,E1 -4534.851,E2 -4534.851} C_VEL
LIN {X 0,Y 530.957,Z 132.343,A -85,B 0,C 180,E1 -4537.509,E2 -4537.509} C_VEL
LIN {X 0,Y 530.944,Z 132.347,A -85,B 0,C 180,E1 -4540.437,E2 -4540.437} C_VEL
LIN {X 0,Y 530.93,Z 132.345,A -85,B 0,C 180,E1 -4543.524,E2 -4543.524} C_VEL
LIN {X 0,Y 530.26,Z 132.431,A -85,B 0,C 180,E1 -4544.158,E2 -4544.158} C_VEL
LIN {X 0,Y 527.416,Z 132.791,A -85,B 0,C 180,E1 -4545.187,E2 -4545.187} C_VEL
LIN {X 0,Y 525.013,Z 133.094,A -85,B 0,C 180,E1 -4546.015,E2 -4546.015} C_VEL
LIN {X 0,Y 523.98,Z 133.22,A -85,B 0,C 180,E1 -4546.655,E2 -4546.655} C_VEL
LIN {X 0,Y 523.895,Z 133.227,A -85,B 0,C 180,E1 -4546.872,E2 -4546.872} C_VEL
LIN {X 0,Y 523.934,Z 133.217,A -85,B 0,C 180,E1 -4549.871,E2 -4549.871} C_VEL
LIN {X 0,Y 523.901,Z 133.224,A -85,B 0,C 180,E1 -4552.868,E2 -4552.868} C_VEL
LIN {X 0,Y 523.928,Z 133.218,A -85,B 0,C 180,E1 -4555.711,E2 -4555.711} C_VEL
LIN {X 0,Y 523.916,Z 133.226,A -85,B 0,C 180,E1 -4558.457,E2 -4558.457} C_VEL
LIN {X 0,Y 523.907,Z 133.22,A -85,B 0,C 180,E1 -4561.124,E2 -4561.124} C_VEL
LIN {X 0,Y 523.919,Z 133.224,A -85,B 0,C 180,E1 -4563.996,E2 -4563.996} C_VEL
LIN {X 0,Y 523.908,Z 133.227,A -85,B 0,C 180,E1 -4566.27,E2 -4566.27} C_VEL
LIN {X 0,Y 523.945,Z 133.219,A -85,B 0,C 180,E1 -4568.767,E2 -4568.767} C_VEL
LIN {X 0,Y 524.033,Z 133.28,A -85,B 0,C 180,E1 -4570.261,E2 -4570.261} C_VEL
LIN {X 0,Y 524.54,Z 138.192,A -85,B 0,C 180,E1 -4571.243,E2 -4571.243} C_VEL
LIN {X 0,Y 524.241,Z 153.981,A -85,B 0,C 180,E1 -4574.249,E2 -4574.249} C_VEL
LIN {X 0,Y 524.253,Z 157.49,A -85,B 0,C 180,E1 -4574.902,E2 -4574.902} C_VEL
LIN {X 0,Y 525.968,Z 166.601,A -85,B 0,C 180,E1 -4575.08,E2 -4575.08} C_VEL
LIN {X 0,Y 525.555,Z 264.574,A -85,B 0,C 180,E1 -4576.442,E2 -4576.442} C_VEL
LIN {X 0,Y 525.391,Z 277.74,A -85,B 0,C 180,E1 -4576.783,E2 -4576.783} C_VEL
LIN {X 0,Y 525.15,Z 289.829,A -85,B 0,C 180,E1 -4577.244,E2 -4577.244} C_VEL
LIN {X 0,Y 524.946,Z 300.324,A -85,B 0,C 180,E1 -4577.777,E2 -4577.777} C_VEL
LIN {X 0,Y 524.741,Z 311.605,A -85,B 0,C 180,E1 -4578.509,E2 -4578.509} C_VEL
LIN {X 0,Y 524.42,Z 322.293,A -85,B 0,C 180,E1 -4579.382,E2 -4579.382} C_VEL
LIN {X 0,Y 524.14,Z 331.906,A -85,B 0,C 180,E1 -4580.352,E2 -4580.352} C_VEL
LIN {X 0,Y 523.925,Z 339.778,A -85,B 0,C 180,E1 -4581.321,E2 -4581.321} C_VEL
LIN {X 0,Y 523.727,Z 347.475,A -85,B 0,C 180,E1 -4582.483,E2 -4582.483} C_VEL
LIN {X 0,Y 523.61,Z 354.531,A -85,B 0,C 180,E1 -4583.836,E2 -4583.836} C_VEL
LIN {X 0,Y 523.406,Z 359.238,A -85,B 0,C 180,E1 -4584.993,E2 -4584.993} C_VEL
LIN {X 0,Y 523.446,Z 362.837,A -85,B 0,C 180,E1 -4586.151,E2 -4586.151} C_VEL
LIN {X 0,Y 523.446,Z 364.698,A -85,B 0,C 180,E1 -4586.922,E2 -4586.922} C_VEL
LIN {X 0,Y 523.338,Z 366.106,A -85,B 0,C 180,E1 -4587.692,E2 -4587.692} C_VEL
LIN {X 0,Y 523.261,Z 367.723,A -85,B 0,C 180,E1 -4589.231,E2 -4589.231} C_VEL
LIN {X 0,Y 523.261,Z 367.96,A -85,B 0,C 180,E1 -4590,E2 -4590} C_VEL
LIN {X 0,Y 523.26,Z 367.777,A -85,B 0,C 180,E1 -4590.77,E2 -4590.77} C_VEL
LIN {X 0,Y 523.338,Z 366.232,A -85,B 0,C 180,E1 -4592.309,E2 -4592.309} C_VEL
LIN {X 0,Y 523.447,Z 364.878,A -85,B 0,C 180,E1 -4593.079,E2 -4593.079} C_VEL
LIN {X 0,Y 523.466,Z 362.023,A -85,B 0,C 180,E1 -4594.235,E2 -4594.235} C_VEL
LIN {X 0,Y 523.465,Z 358.152,A -85,B 0,C 180,E1 -4595.393,E2 -4595.393} C_VEL
LIN {X 0,Y 523.567,Z 352.82,A -85,B 0,C 180,E1 -4596.622,E2 -4596.622} C_VEL
LIN {X 0,Y 523.786,Z 345.639,A -85,B 0,C 180,E1 -4597.905,E2 -4597.905} C_VEL
LIN {X 0,Y 523.967,Z 337.504,A -85,B 0,C 180,E1 -4599.068,E2 -4599.068} C_VEL
LIN {X 0,Y 524.213,Z 329.173,A -85,B 0,C 180,E1 -4600.037,E2 -4600.037} C_VEL
LIN {X 0,Y 524.523,Z 318.888,A -85,B 0,C 180,E1 -4601.008,E2 -4601.008} C_VEL
LIN {X 0,Y 524.774,Z 308.305,A -85,B 0,C 180,E1 -4601.812,E2 -4601.812} C_VEL
LIN {X 0,Y 525.052,Z 297.548,A -85,B 0,C 180,E1 -4602.465,E2 -4602.465} C_VEL
LIN {X 0,Y 525.281,Z 285.028,A -85,B 0,C 180,E1 -4603.049,E2 -4603.049} C_VEL
LIN {X 0,Y 525.486,Z 272.493,A -85,B 0,C 180,E1 -4603.462,E2 -4603.462} C_VEL
LIN {X 0,Y 525.664,Z 259.732,A -85,B 0,C 180,E1 -4603.728,E2 -4603.728} C_VEL
LIN {X 0,Y 525.842,Z 166.196,A -85,B 0,C 180,E1 -4605.02,E2 -4605.02} C_VEL
LIN {X 0,Y 524.219,Z 157.404,A -85,B 0,C 180,E1 -4605.206,E2 -4605.206} C_VEL
LIN {X 0,Y 524.49,Z 141.77,A -85,B 0,C 180,E1 -4608.152,E2 -4608.152} C_VEL
LIN {X 0,Y 524.475,Z 136.567,A -85,B 0,C 180,E1 -4609.166,E2 -4609.166} C_VEL
LIN {X 0,Y 524.035,Z 133.213,A -85,B 0,C 180,E1 -4609.89,E2 -4609.89} C_VEL
LIN {X 0,Y 523.911,Z 133.22,A -85,B 0,C 180,E1 -4612.894,E2 -4612.894} C_VEL
LIN {X 0,Y 523.908,Z 133.223,A -85,B 0,C 180,E1 -4615.421,E2 -4615.421} C_VEL
LIN {X 0,Y 523.917,Z 133.225,A -85,B 0,C 180,E1 -4618.002,E2 -4618.002} C_VEL
LIN {X 0,Y 523.937,Z 133.216,A -85,B 0,C 180,E1 -4620.853,E2 -4620.853} C_VEL
LIN {X 0,Y 523.96,Z 133.222,A -85,B 0,C 180,E1 -4623.734,E2 -4623.734} C_VEL
LIN {X 0,Y 523.899,Z 133.221,A -85,B 0,C 180,E1 -4626.4,E2 -4626.4} C_VEL
LIN {X 0,Y 523.913,Z 133.222,A -85,B 0,C 180,E1 -4629.085,E2 -4629.085} C_VEL
LIN {X 0,Y 523.94,Z 133.217,A -85,B 0,C 180,E1 -4632.12,E2 -4632.12} C_VEL
LIN {X 0,Y 523.938,Z 133.225,A -85,B 0,C 180,E1 -4635.31,E2 -4635.31} C_VEL
LIN {X 0,Y 523.938,Z 133.218,A -85,B 0,C 180,E1 -4638.692,E2 -4638.692} C_VEL
LIN {X 0,Y 523.911,Z 133.22,A -85,B 0,C 180,E1 -4641.898,E2 -4641.898} C_VEL
LIN {X 0,Y 523.916,Z 133.225,A -85,B 0,C 180,E1 -4644.912,E2 -4644.912} C_VEL
LIN {X 0,Y 523.928,Z 133.218,A -85,B 0,C 180,E1 -4647.68,E2 -4647.68} C_VEL
LIN {X 0,Y 523.933,Z 133.222,A -85,B 0,C 180,E1 -4650.68,E2 -4650.68} C_VEL
LIN {X 0,Y 523.93,Z 133.217,A -85,B 0,C 180,E1 -4653.726,E2 -4653.726} C_VEL
LIN {X 0,Y 523.905,Z 133.223,A -85,B 0,C 180,E1 -4656.269,E2 -4656.269} C_VEL
LIN {X 0,Y 523.941,Z 133.223,A -85,B 0,C 180,E1 -4658.766,E2 -4658.766} C_VEL
LIN {X 0,Y 523.924,Z 133.219,A -85,B 0,C 180,E1 -4661.22,E2 -4661.22} C_VEL
LIN {X 0,Y 523.907,Z 133.228,A -85,B 0,C 180,E1 -4664.437,E2 -4664.437} C_VEL
LIN {X 0,Y 523.948,Z 133.215,A -85,B 0,C 180,E1 -4667.607,E2 -4667.607} C_VEL
LIN {X 0,Y 523.926,Z 133.221,A -85,B 0,C 180,E1 -4669.957,E2 -4669.957} C_VEL
LIN {X 0,Y 523.988,Z 133.21,A -85,B 0,C 180,E1 -4673.067,E2 -4673.067} C_VEL
LIN {X 0,Y 523.942,Z 133.216,A -85,B 0,C 180,E1 -4675.384,E2 -4675.384} C_VEL
LIN {X 0,Y 524.099,Z 133.199,A -85,B 0,C 180,E1 -4677.694,E2 -4677.694} C_VEL
LIN {X 0,Y 524.092,Z 133.205,A -85,B 0,C 180,E1 -4680,E2 -4680} C_VEL
LIN {X 0,Y 524.099,Z 133.201,A -85,B 0,C 180,E1 -4682.306,E2 -4682.306} C_VEL
LIN {X 0,Y 523.995,Z 133.214,A -85,B 0,C 180,E1 -4686.16,E2 -4686.16} C_VEL
LIN {X 0,Y 523.938,Z 133.218,A -85,B 0,C 180,E1 -4689.263,E2 -4689.263} C_VEL
LIN {X 0,Y 523.915,Z 133.22,A -85,B 0,C 180,E1 -4692.394,E2 -4692.394} C_VEL
LIN {X 0,Y 523.879,Z 133.231,A -85,B 0,C 180,E1 -4695.564,E2 -4695.564} C_VEL
LIN {X 0,Y 523.905,Z 133.223,A -85,B 0,C 180,E1 -4697.971,E2 -4697.971} C_VEL
LIN {X 0,Y 523.911,Z 133.219,A -85,B 0,C 180,E1 -4700.413,E2 -4700.413} C_VEL
LIN {X 0,Y 523.88,Z 133.225,A -85,B 0,C 180,E1 -4702.895,E2 -4702.895} C_VEL
LIN {X 0,Y 523.892,Z 133.23,A -85,B 0,C 180,E1 -4705.422,E2 -4705.422} C_VEL
LIN {X 0,Y 523.892,Z 133.222,A -85,B 0,C 180,E1 -4708.003,E2 -4708.003} C_VEL
LIN {X 0,Y 523.894,Z 133.225,A -85,B 0,C 180,E1 -4710.846,E2 -4710.846} C_VEL
LIN {X 0,Y 523.923,Z 133.219,A -85,B 0,C 180,E1 -4713.729,E2 -4713.729} C_VEL
LIN {X 0,Y 523.885,Z 133.224,A -85,B 0,C 180,E1 -4716.399,E2 -4716.399} C_VEL
LIN {X 0,Y 523.909,Z 133.227,A -85,B 0,C 180,E1 -4719.086,E2 -4719.086} C_VEL
LIN {X 0,Y 523.897,Z 133.222,A -85,B 0,C 180,E1 -4722.125,E2 -4722.125} C_VEL
LIN {X 0,Y 523.933,Z 133.219,A -85,B 0,C 180,E1 -4725.312,E2 -4725.312} C_VEL
LIN {X 0,Y 523.919,Z 133.228,A -85,B 0,C 180,E1 -4728.695,E2 -4728.695} C_VEL
LIN {X 0,Y 523.91,Z 133.22,A -85,B 0,C 180,E1 -4731.898,E2 -4731.898} C_VEL
LIN {X 0,Y 523.917,Z 133.222,A -85,B 0,C 180,E1 -4734.913,E2 -4734.913} C_VEL
LIN {X 0,Y 523.934,Z 133.217,A -85,B 0,C 180,E1 -4737.68,E2 -4737.68} C_VEL
LIN {X 0,Y 523.937,Z 133.222,A -85,B 0,C 180,E1 -4740.68,E2 -4740.68} C_VEL
LIN {X 0,Y 523.904,Z 133.225,A -85,B 0,C 180,E1 -4743.725,E2 -4743.725} C_VEL
LIN {X 0,Y 523.946,Z 133.291,A -85,B 0,C 180,E1 -4745.48,E2 -4745.48} C_VEL
LIN {X 0,Y 525.311,Z 140.92,A -85,B 0,C 180,E1 -4746.754,E2 -4746.754} C_VEL
LIN {X 0,Y 525.074,Z 155.371,A -85,B 0,C 180,E1 -4749.02,E2 -4749.02} C_VEL
LIN {X 0,Y 524.561,Z 176.331,A -85,B 0,C 180,E1 -4752.254,E2 -4752.254} C_VEL
LIN {X 0,Y 524.213,Z 193.154,A -85,B 0,C 180,E1 -4754.819,E2 -4754.819} C_VEL
LIN {X 0,Y 525.884,Z 205.29,A -85,B 0,C 180,E1 -4755.054,E2 -4755.054} C_VEL
LIN {X 0,Y 525.522,Z 301.641,A -85,B 0,C 180,E1 -4756.391,E2 -4756.391} C_VEL
LIN {X 0,Y 525.31,Z 314.935,A -85,B 0,C 180,E1 -4756.73,E2 -4756.73} C_VEL
LIN {X 0,Y 524.969,Z 328.237,A -85,B 0,C 180,E1 -4757.238,E2 -4757.238} C_VEL
LIN {X 0,Y 524.726,Z 340.477,A -85,B 0,C 180,E1 -4757.888,E2 -4757.888} C_VEL
LIN {X 0,Y 524.461,Z 352.319,A -85,B 0,C 180,E1 -4758.698,E2 -4758.698} C_VEL
LIN {X 0,Y 524.158,Z 362.528,A -85,B 0,C 180,E1 -4759.571,E2 -4759.571} C_VEL
LIN {X 0,Y 523.935,Z 371.717,A -85,B 0,C 180,E1 -4760.542,E2 -4760.542} C_VEL
LIN {X 0,Y 523.716,Z 380.673,A -85,B 0,C 180,E1 -4761.705,E2 -4761.705} C_VEL
LIN {X 0,Y 523.568,Z 387.882,A -85,B 0,C 180,E1 -4762.867,E2 -4762.867} C_VEL
LIN {X 0,Y 523.46,Z 392.747,A -85,B 0,C 180,E1 -4763.834,E2 -4763.834} C_VEL
LIN {X 0,Y 523.383,Z 397.476,A -85,B 0,C 180,E1 -4764.992,E2 -4764.992} C_VEL
LIN {X 0,Y 523.443,Z 401.094,A -85,B 0,C 180,E1 -4766.15,E2 -4766.15} C_VEL
LIN {X 0,Y 523.367,Z 402.956,A -85,B 0,C 180,E1 -4766.921,E2 -4766.921} C_VEL
